//--------------------------------------------------------------------------------------------------------------------------------------------------------------------------------
3014://Comanda para posição de mesa de giro final após eixo X se movimentar 20% do trajeto para garantir que não colida a mesa de giro com a esteira de inspeção

	IF LA_GERAL.bit_MAQUINA_RODANDO AND (LA_EMP.info_MOTOR_EIXO_X_EMPILHADOR_POS_ATUAL > 130 AND LA_EMP.info_MOTOR_EIXO_X_EMPILHADOR_POS_ATUAL < 780) THEN
		LA_EMP.bit_EIXO_GIRO_MESA_MOVER_ABS		:= TRUE;
		
		passo_X_EMPILHADOR 									:= 3015;
	END_IF
	
//--------------------------------------------------------------------------------------------------------------------------------------------------------------------------------
3015: //verifica se a mesa de giro está se movendo para posição final. Caso esteja, desativa comando de movimento absoluto

	IF	M2_LA_EMP_GIRO.bit_MOVE_ABS_FAZENDO OR LA_EMP.bit_EIXO_GIRO_MESA_POSICIONADO	THEN
			LA_EMP.bit_EIXO_GIRO_MESA_MOVER_ABS	:= FALSE;
			passo_X_EMPILHADOR 								:= 3016;
	END_IF
	
//--------------------------------------------------------------------------------------------------------------------------------------------------------------------------------
3016: //verifica se a mesa de giro completou movimento

	IF	M2_LA_EMP_GIRO.bit_MOVE_ABS_FEITO OR LA_EMP.bit_EIXO_GIRO_MESA_POSICIONADO	THEN
			LA_EMP.bit_MESA_GIRO_CONCLUIDO	:= TRUE;
			passo_X_EMPILHADOR 							:= 3017;
	END_IF	
	
//--------------------------------------------------------------------------------------------------------------------------------------------------------------------------------
3017: //aguarda liberação da sacola depositada na mesa para liberar movimento do eixo X da empilhadora para próxima posição de pega	
	
// 	IF 		(PVAR.rec_ATUAL.int_NUM_MAX_CAMADAS_EMPILHADOR - 4) = 0 	THEN
// 				passo_X_EMPILHADOR			:= 3028;
// 	ELSIF 	(PVAR.rec_ATUAL.int_NUM_MAX_CAMADAS_EMPILHADOR - 4) = 1		THEN
// 				passo_X_EMPILHADOR			:= 3018;
// 		
// 	END_IF	

	IF 	(PVAR.rec_ATUAL.int_NUM_MAX_CAMADAS_EMPILHADOR - 4) = 0 	THEN
		M2_LA_EMP_GIRO.ABS_MOVER			:= PVAR.rec_ATUAL.coord_MESA_GIRO_INICIAL;
	END_IF

	passo_X_EMPILHADOR			:= 3018;
	
	
//--------------------------------------------------------------------------------------------------------------------------------------------------------------------------------
3018: //manda os valores de coordenada para movimentos absolutos da posição 9 do eixo X e declara que está na posição 9

	IF LA_EMP.bit_ENTREGA_EMPILHADOR_CONCLUIDO THEN
		M0_LA_EMP_X.ABS_MOVER	:= PVAR.rec_ATUAL.coord_X_EMPILHADOR_POS[PVAR.rec_ATUAL.int_NUM_MAX_CAMADAS_EMPILHADOR - 3];
		PVAR.int_POSICAO_EIXO_X_EMPILHADOR	:=	9;
		passo_X_EMPILHADOR 					:= 3019;
	END_IF
	
//--------------------------------------------------------------------------------------------------------------------------------------------------------------------------------
3019: // Comanda eixo X do empilhador com movimento absoluto para posição 9.

	IF LA_GERAL.bit_MAQUINA_RODANDO  THEN
		LA_EMP.bit_EIXO_X_EMPILHADOR_MOVER_ABS	:= TRUE;
		LA_EMP.bit_EIXO_GIRO_MESA_MOVER_ABS		:= TRUE;
		passo_X_EMPILHADOR 									:= 3020;	
	END_IF
	
//--------------------------------------------------------------------------------------------------------------------------------------------------------------------------------
3020: //verifica se o eixo X do empilhador está se movendo para posição 9. Caso esteja, desativa comando de movimento absoluto

	IF	M0_LA_EMP_X.bit_MOVE_ABS_FAZENDO OR LA_EMP.bit_EIXO_X_EMPILHADOR_POSICIONADO	THEN
			LA_EMP.bit_EIXO_X_EMPILHADOR_MOVER_ABS	:= FALSE;
			LA_EMP.bit_EIXO_GIRO_MESA_MOVER_ABS		:= FALSE;
			passo_X_EMPILHADOR 									:= 3021;
	END_IF
	
	
//--------------------------------------------------------------------------------------------------------------------------------------------------------------------------------
3021: //verifica se o eixo X do empilhador completou movimento

	IF	M0_LA_EMP_X.bit_MOVE_ABS_FEITO OR LA_EMP.bit_EIXO_X_EMPILHADOR_POSICIONADO	THEN
			LA_EMP.bit_LIBERA_PEGA			:= TRUE;
			passo_X_EMPILHADOR							:= 3022;
	END_IF


//--------------------------------------------------------------------------------------------------------------------------------------------------------------------------------
3022: //aguarda liberação da sacola depositada na mesa para liberar movimento do eixo X da empilhadora para POSIÇÃO 1

	IF 		(PVAR.rec_ATUAL.int_NUM_MAX_CAMADAS_EMPILHADOR - 4) = 0 		THEN
				passo_X_EMPILHADOR			:= 3025;
	ELSE		
				passo_X_EMPILHADOR			:= 3023;
	END_IF
	
//--------------------------------------------------------------------------------------------------------------------------------------------------------------------------------
3023: //manda os valores de coordenada para movimentos absolutos da posição 10 do eixo X e declara que está na posição 10

	IF LA_EMP.bit_ENTREGA_EMPILHADOR_CONCLUIDO THEN
		M0_LA_EMP_X.ABS_MOVER	:= PVAR.rec_ATUAL.coord_X_EMPILHADOR_POS[1];
		M2_LA_EMP_GIRO.ABS_MOVER			:= PVAR.rec_ATUAL.coord_MESA_GIRO_INICIAL;
		PVAR.int_POSICAO_EIXO_X_EMPILHADOR	:=	10;
		passo_X_EMPILHADOR 					:= 3024;
	END_IF
	
	// 	IF tmr_passo_3021.Q	THEN
	// 		passo_X_EMPILHADOR 					:= 3021;
	// 	END_IF
	
	
//--------------------------------------------------------------------------------------------------------------------------------------------------------------------------------
3024: // Comanda eixo X do empilhador com movimento absoluto para posição 10.

	IF LA_GERAL.bit_MAQUINA_RODANDO  THEN
		LA_EMP.bit_EIXO_X_EMPILHADOR_MOVER_ABS	:= TRUE;
		LA_EMP.bit_EIXO_GIRO_MESA_MOVER_ABS		:= TRUE;
		passo_X_EMPILHADOR 									:= 3025;	
	END_IF
	
//--------------------------------------------------------------------------------------------------------------------------------------------------------------------------------
3025: //verifica se o eixo X do empilhador está se movendo para posição 10. Caso esteja, desativa comando de movimento absoluto

	IF	M0_LA_EMP_X.bit_MOVE_ABS_FAZENDO OR LA_EMP.bit_EIXO_X_EMPILHADOR_POSICIONADO	THEN
			LA_EMP.bit_EIXO_X_EMPILHADOR_MOVER_ABS	:= FALSE;
			passo_X_EMPILHADOR 									:= 3026;
	END_IF
	
//--------------------------------------------------------------------------------------------------------------------------------------------------------------------------------
3026: //verifica se o eixo rotativo do empilhador está se movendo para posição inicial. Caso esteja, desativa comando de movimento absoluto

	IF	M2_LA_EMP_GIRO.bit_MOVE_ABS_FAZENDO OR LA_EMP.bit_EIXO_GIRO_MESA_POSICIONADO	THEN
			LA_EMP.bit_EIXO_GIRO_MESA_MOVER_ABS		:= FALSE;
			passo_X_EMPILHADOR 									:= 3027;
	END_IF
	
//--------------------------------------------------------------------------------------------------------------------------------------------------------------------------------
3027: //verifica se o eixo X do empilhador completou movimento	
	
	IF	M0_LA_EMP_X.bit_MOVE_ABS_FEITO	OR 	LA_EMP.bit_EIXO_X_EMPILHADOR_POSICIONADO	THEN
			bit_X_EMPILHADOR_FEITO				:= TRUE;
			LA_EMP.bit_LIBERA_PEGA	:= TRUE;
	END_IF	
	
	IF	M2_LA_EMP_GIRO.bit_MOVE_ABS_FEITO	OR 	LA_EMP.bit_EIXO_GIRO_MESA_POSICIONADO	THEN
			bit_GIRO_MESA_FEITO	:= TRUE;
	END_IF	
	
	IF	bit_X_EMPILHADOR_FEITO		AND
		bit_GIRO_MESA_FEITO			THEN
			bit_X_EMPILHADOR_FEITO		:= FALSE;
			bit_GIRO_MESA_FEITO			:= FALSE;
		
			passo_X_EMPILHADOR 			:= 3028;
	END_IF		
	
//--------------------------------------------------------------------------------------------------------------------------------------------------------------------------------
3028://aguarda confirmação de pilha entregue e comanda posições para entregar pilha para inspeção

	M0_LA_EMP_X.ABS_MOVER		 	:= PVAR.rec_ATUAL.coord_X_EMPILHADOR_INSPECAO;
	M2_LA_EMP_GIRO.ABS_MOVER		 			:= PVAR.rec_ATUAL.coord_MESA_GIRO_INSPECAO;
	LA_EMP.bit_REALIZANDO_INSPECAO 	:= TRUE;
	passo_X_EMPILHADOR							:= 3029;
	
//--------------------------------------------------------------------------------------------------------------------------------------------------------------------------------
3029://comanda movimento da mesa de giro para posição de inspeção

	LA_EMP.bit_LIBERA_PEGA	:= FALSE;

	IF LA_GERAL.bit_MAQUINA_RODANDO AND LA_EMP.bit_ENTREGA_EMPILHADOR_CONCLUIDO	THEN
		LA_EMP.bit_EIXO_GIRO_MESA_MOVER_ABS		:= TRUE;
		passo_X_EMPILHADOR									:= 3030;
	END_IF

//--------------------------------------------------------------------------------------------------------------------------------------------------------------------------------
3030: //verifica se o eixo rotativo do empilhador está se movendo para posição inicial. Caso esteja, desativa comando de movimento absoluto

	IF	M2_LA_EMP_GIRO.bit_MOVE_ABS_FAZENDO OR LA_EMP.bit_EIXO_GIRO_MESA_POSICIONADO	THEN
			LA_EMP.bit_EIXO_GIRO_MESA_MOVER_ABS		:= FALSE;
			passo_X_EMPILHADOR 									:= 3031;
	END_IF	
	
//--------------------------------------------------------------------------------------------------------------------------------------------------------------------------------
3031://verifica se a mesa de giro completou o movimento	

	IF	M2_LA_EMP_GIRO.bit_MOVE_ABS_FEITO OR LA_EMP.bit_EIXO_GIRO_MESA_POSICIONADO	THEN
			passo_X_EMPILHADOR 	:= 3032;
	END_IF

//--------------------------------------------------------------------------------------------------------------------------------------------------------------------------------
3032://se a máquina estiver rodando, comanda movimento do eixo X do empilhador para inspeção

	IF LA_GERAL.bit_MAQUINA_RODANDO	THEN
		LA_EMP.bit_EIXO_X_EMPILHADOR_MOVER_ABS	:= TRUE;
		passo_X_EMPILHADOR 									:= 3033;
	END_IF
	
//--------------------------------------------------------------------------------------------------------------------------------------------------------------------------------
3033://verifica se o eixo X do empilhador está se movendo para inspeção. Caso esteja, desativa comando de movimento absoluto

	IF	M0_LA_EMP_X.bit_MOVE_ABS_FAZENDO OR LA_EMP.bit_EIXO_X_EMPILHADOR_POSICIONADO	THEN
			LA_EMP.bit_EIXO_X_EMPILHADOR_MOVER_ABS	:= FALSE;
			passo_X_EMPILHADOR 									:= 3034;
	END_IF	
	
//--------------------------------------------------------------------------------------------------------------------------------------------------------------------------------
3034: // verifica se eixo X do empilhador completou movimento

	IF	M0_LA_EMP_X.bit_MOVE_ABS_FEITO OR  LA_EMP.bit_EIXO_X_EMPILHADOR_POSICIONADO	THEN
		LA_EMP.bit_LIBERA_INSPECAO_PILHA		:= 	TRUE;
		passo_X_EMPILHADOR 								:= 3035;
	END_IF	

	
//--------------------------------------------------------------------------------------------------------------------------------------------------------------------------------
3035://liga esteira de mesa giro para liberar pilha de sacola para esteira de inspeção
	
	LA_EMP.est_ROLETES_GIRO_MESA_REVERSE	:= FALSE;
	LA_EMP.est_ROLETES_GIRO_MESA			:= TRUE;
	passo_X_EMPILHADOR 								:= 3036;
	
//--------------------------------------------------------------------------------------------------------------------------------------------------------------------------------
3036://Após um tempo fora do sensor de presença da mesa de giro, considera que a pilha saiu da mesa de giro e conclui processo de entrega para mesa de inspeção
	

	IF LA_EMP.di_SENS_EST_INSPEC_PRODUTO_2 AND NOT LA_EMP.di_SENS_PRODUTO_MESA_GIRO THEN
		bit_RESET_CONTAGEM		:= TRUE;
		passo_X_EMPILHADOR 		:= 3037;
	END_IF
	
	
//--------------------------------------------------------------------------------------------------------------------------------------------------------------------------------
3037://Declara pilha como entregue e para a esteira da mesa giro. Prepara mesa de giro para posição de reinicio

	tmr_sens_MESA_GIRO_IN.IN						:= FALSE;
	LA_EMP.est_ROLETES_GIRO_MESA			:= FALSE;
	LA_EMP.est_ROLETES_GIRO_MESA_REVERSE	:= FALSE;
	
	LA_EMP.bit_EST_PILHA_ENTREGUE		 	:= FALSE;
	LA_EMP.bit_LIBERA_INSPECAO_PILHA	 	:= FALSE;
	LA_EMP.bit_EST_INSPECAO_ENTREGUE_1 	:= FALSE;
	LA_EMP.bit_EST_INSPECAO_ENTREGUE_2 	:= FALSE;
	bit_RESET_CONTAGEM							 	:= FALSE;
	LA_EMP.bit_REALIZANDO_INSPECAO	 	:= FALSE;
	LA_EMP.bit_valv_DESCE_MESA_GIRO	 	:= FALSE;

	passo_X_EMPILHADOR							 	:= 998;
	

	
END_CASE

//--------------------------------------------------------------------------------------------------------------------------------------------------------------------------------
//--------------------------------------------------------------------------------------------------------------------------------------------------------------------------------
//LÓGICAS AUXILIARES


	
	
(*//CONTINUAR MOVIMENTO DO EIXO X DO EMPILHADOR APÓS PARADA DE EMERGÊNCIA
	IF (bt_MAQUINA_RESET OR bt_MAQUINA_RESET_2) AND NOT GVL_CELULA.bit_MAQUINA_RODANDO	THEN
			
			IF 	passo_X_EMPILHADOR >= 0 	AND
				passo_X_EMPILHADOR <= 15 	THEN
				GVL_EMPILHAMENTO.bit_EIXO_X_EMPILHADOR_MOVER_ABS		:= FALSE;
				passo_X_EMPILHADOR := 9;
			END_IF	
	
			IF 	(passo_X_EMPILHADOR >= 1000	AND
				passo_X_EMPILHADOR <= 1003) THEN
				GVL_EMPILHAMENTO.bit_EIXO_X_EMPILHADOR_MOVER_ABS		:= FALSE;
				passo_X_EMPILHADOR := 999;
			END_IF
			
			IF 	passo_X_EMPILHADOR >= 1005 	AND
				passo_X_EMPILHADOR <= 1008 	THEN
				GVL_EMPILHAMENTO.bit_EIXO_X_EMPILHADOR_MOVER_ABS		:= FALSE;
				passo_X_EMPILHADOR := 1005;
			END_IF
			
			IF 	passo_X_EMPILHADOR >= 1010 	AND
				passo_X_EMPILHADOR <= 1013 	THEN
				GVL_EMPILHAMENTO.bit_EIXO_X_EMPILHADOR_MOVER_ABS		:= FALSE;
				passo_X_EMPILHADOR := 1010;
			END_IF
			
			IF 	passo_X_EMPILHADOR >= 1015 	AND
				passo_X_EMPILHADOR <= 1018 	THEN
				GVL_EMPILHAMENTO.bit_EIXO_X_EMPILHADOR_MOVER_ABS		:= FALSE;
				passo_X_EMPILHADOR := 1015;
			END_IF
			
			IF 	passo_X_EMPILHADOR >= 1020 	AND
				passo_X_EMPILHADOR <= 1023 	THEN
				GVL_EMPILHAMENTO.bit_EIXO_X_EMPILHADOR_MOVER_ABS		:= FALSE;
				passo_X_EMPILHADOR := 1020;
			END_IF
			
			IF 	passo_X_EMPILHADOR >= 1025 	AND
				passo_X_EMPILHADOR <= 1028 	THEN
				GVL_EMPILHAMENTO.bit_EIXO_X_EMPILHADOR_MOVER_ABS		:= FALSE;
				passo_X_EMPILHADOR := 1025;
			END_IF
			
			IF 	passo_X_EMPILHADOR >= 2000 	AND
				passo_X_EMPILHADOR <= 2003	THEN
				GVL_EMPILHAMENTO.bit_EIXO_X_EMPILHADOR_MOVER_ABS		:= FALSE;
				passo_X_EMPILHADOR := 2000;
			END_IF
			
			IF 	passo_X_EMPILHADOR >= 2005 	AND
				passo_X_EMPILHADOR <= 2008	THEN
				GVL_EMPILHAMENTO.bit_EIXO_X_EMPILHADOR_MOVER_ABS		:= FALSE;
				passo_X_EMPILHADOR := 2005;
			END_IF
			
			IF 	passo_X_EMPILHADOR >= 2010 	AND
				passo_X_EMPILHADOR <= 2013	THEN
				GVL_EMPILHAMENTO.bit_EIXO_X_EMPILHADOR_MOVER_ABS		:= FALSE;
				passo_X_EMPILHADOR := 2010;
			END_IF
			
			IF 	passo_X_EMPILHADOR >= 2015 	AND
				passo_X_EMPILHADOR <= 2015	THEN
				GVL_EMPILHAMENTO.bit_EIXO_X_EMPILHADOR_MOVER_ABS		:= FALSE;
				passo_X_EMPILHADOR := 2015;
			END_IF
			
			IF 	passo_X_EMPILHADOR >= 2020 	AND
				passo_X_EMPILHADOR <= 2023	THEN
				GVL_EMPILHAMENTO.bit_EIXO_X_EMPILHADOR_MOVER_ABS		:= FALSE;
				passo_X_EMPILHADOR := 2020;
			END_IF
			
	END_IF
	
*)

	
	
	//EIXO X EMPILHADOR JÁ ESTÁ NA POSIÇÃO
	IF	LA_EMP.info_MOTOR_EIXO_X_EMPILHADOR_POS_ATUAL	>= M0_LA_EMP_X.ABS_MOVER.sp_POSICAO - 1	AND
		LA_EMP.info_MOTOR_EIXO_X_EMPILHADOR_POS_ATUAL	<= M0_LA_EMP_X.ABS_MOVER.sp_POSICAO + 1	THEN
			LA_EMP.bit_EIXO_X_EMPILHADOR_POSICIONADO	:= TRUE;
	ELSE
			LA_EMP.bit_EIXO_X_EMPILHADOR_POSICIONADO	:= FALSE;
	END_IF
	
	
	//EIXO X EMPILHADOR JÁ ESTÁ NA POSIÇÃO
	IF	LA_EMP.info_MOTOR_GIRO_MESA_POS_ATUAL	>= M2_LA_EMP_GIRO.ABS_MOVER.sp_POSICAO - 1	AND
		LA_EMP.info_MOTOR_GIRO_MESA_POS_ATUAL	<= M2_LA_EMP_GIRO.ABS_MOVER.sp_POSICAO + 1	THEN
			LA_EMP.bit_EIXO_GIRO_MESA_POSICIONADO	:= TRUE;
	ELSE
			LA_EMP.bit_EIXO_GIRO_MESA_POSICIONADO	:= FALSE;
	END_IF
	
	
		
	//Define se a posicão da mesa de giro de acordo com a posição atual do eixo X
	IF M2_LA_EMP_GIRO.ABS_MOVER.sp_POSICAO > 90 THEN
		LA_EMP.bit_GIRO_MESA_FOWARD	:=	TRUE;
		LA_EMP.bit_GIRO_MESA_REVERSE	:=	FALSE;
	ELSE
		LA_EMP.bit_GIRO_MESA_FOWARD	:=	FALSE;
		LA_EMP.bit_GIRO_MESA_REVERSE	:=	TRUE;
	END_IF
	

	
	
//TIMERS EIXO X
tmr_HOME 	  (PT	:= T#200MS);
tmr_ENTREGA_X (PT	:= T#100MS);
tmr_passo_2021(PT	:= T#300MS);
tmr_passo_2032(PT	:= T#500MS);
tmr_LIBERA_X_INSPECAO(PT	:= T#1500MS);
cont_PILHA_ENTREGA(CU:= bit_INCREMENTA_SACOLA, RESET:= bit_RESET_CONTAGEM, PV:= 999, CV=> pvar.int_PILHAS_ENTREGUES);	


//TIMERS GIRO MESA
tmr_HOME 			(PT	:= T#200MS);
tmr_sens_MESA_GIRO_IN 	(PT	:= T#500MS);
tmr_sens_MESA_GIRO_OUT 	(PT	:= T#2300MS);
TMR_GIRO_1		 	(PT	:= T#4000MS);
TMR_GIRO_2		 	(PT	:= T#4000MS);
TMR_GIRO_3		 	(PT	:= T#4000MS);
TMR_GIRO_4		 	(PT	:= T#500MS);
TMR_GIRO_5		 	(PT	:= T#4000MS);
TMR_GIRO_10		 	(PT	:= T#4000MS);

tmr_passo_1041		 	(PT	:= T#300MS);

END_PROGRAM

// LADO_A/02 - LA_EMPILHADOR/B03_INSPECAO
PROGRAM B03_INSPECAO
VAR
	passo_INSPECAO		: INT := 9;
	tmr_INSPECAO_OK		: TON;
	tmr_LIBERA_INSPECAO_OK		: TON;
END_VAR

//MOVE O PASSO PARA O HOME

	IF	LA_IHM.bit_bt_RESET_INSPECAO	THEN
			passo_INSPECAO								:= 9;
	END_IF
	
CASE	passo_INSPECAO	OF
	
//--------------------------------------------------------------------------------------------------------------------------------------------------------------------------------
09: //HOME: Reseta variáveis

	IF NOT LA_EMP.di_SENS_EST_INSPEC_PRODUTO_1 AND NOT LA_EMP.di_SENS_EST_INSPEC_PRODUTO_2 THEN
		LA_EMP.bit_OPERADOR_INSPECAO_OK		:=	FALSE;
		LA_EMP.bit_EST_ENVIAR_PILHA_INSPECAO	:=	FALSE;
		LA_EMP.bit_EST_INSPECAO_ENTREGUE_2	:=	FALSE;
		LA_EMP.est_INSPECAO_EMPILHADOR		:= 	FALSE;
		tmr_LIBERA_INSPECAO_OK.IN						:=	FALSE;
		bt_LAMP_INSPECAO_OK 							:=  FALSE;
		passo_INSPECAO									:=  999;
	ELSIF LA_EMP.bit_OPERADOR_INSPECAO_OK THEN
		passo_INSPECAO									:= 1002;
	END_IF
	
	
//--------------------------------------------------------------------------------------------------------------------------------------------------------------------------------
999://aguarda esteira da mesa giro entregar pilha para inspeção e liga esteira

	IF LA_EMP.bit_LIBERA_INSPECAO_PILHA	THEN
		LA_EMP.est_INSPECAO_EMPILHADOR	:= TRUE;
		passo_INSPECAO								:= 1000;
	END_IF
	
	IF LA_EMP.bit_OPERADOR_INSPECAO_OK THEN
		LA_EMP.bit_STATUS_INSPECAO_1		:= FALSE;
		passo_INSPECAO								:= 1002;
	END_IF
	
	
//--------------------------------------------------------------------------------------------------------------------------------------------------------------------------------
1000://espera feedback dos sensores da esteira de inspeção para garantir que a pilha chegou até o fim. 

	IF  LA_EMP.di_SENS_EST_INSPEC_PRODUTO_2 THEN
		LA_EMP.est_INSPECAO_EMPILHADOR		:= FALSE;
		LA_EMP.bit_STATUS_INSPECAO_1			:= TRUE;
		//GVL_EMPILHAMENTO.bit_EST_INSPECAO_ENTREGUE_1	:= TRUE;
		
		passo_INSPECAO									:= 999;
	END_IF
	
	
//--------------------------------------------------------------------------------------------------------------------------------------------------------------------------------
1001://aguarda comando de operador indicando que a pilha está ok para ser devolvida

	IF LA_EMP.bit_OPERADOR_INSPECAO_OK THEN
		LA_EMP.bit_STATUS_INSPECAO_1	:= FALSE;
		passo_INSPECAO							:= 1002;
	END_IF
	
//--------------------------------------------------------------------------------------------------------------------------------------------------------------------------------
1002://espera confirmação de recebimento OK da esteira mesa giro e liga esteira de inspeção reverse para devolução de pilha 

	IF LA_EMP.bit_EST_ENVIAR_PILHA_INSPECAO THEN
		LA_EMP.est_INSPECAO_EMPILHADOR_REVERSE 	:= TRUE;
		LA_EMP.est_INSPECAO_EMPILHADOR			:= TRUE;
		passo_INSPECAO										:= 1003;
	END_IF
	
	
//--------------------------------------------------------------------------------------------------------------------------------------------------------------------------------
1003://ao deixar de receber feedback dos dois sensores da esteira de inspeção, para esteira e reinicia ciclo

	IF NOT LA_EMP.di_SENS_EST_INSPEC_PRODUTO_1 AND NOT LA_EMP.di_SENS_EST_INSPEC_PRODUTO_2 THEN
		tmr_LIBERA_INSPECAO_OK.IN							:= TRUE;
	ELSE
		tmr_LIBERA_INSPECAO_OK.IN							:= FALSE;
	END_IF
	
	IF tmr_LIBERA_INSPECAO_OK.Q	THEN
		passo_INSPECAO										:= 1004;
	END_IF
	
//--------------------------------------------------------------------------------------------------------------------------------------------------------------------------------
1004:
		LA_EMP.est_INSPECAO_EMPILHADOR_REVERSE	:= FALSE;
		LA_EMP.est_INSPECAO_EMPILHADOR			:= FALSE;
		tmr_LIBERA_INSPECAO_OK.IN							:= FALSE;
		LA_EMP.bit_EST_INSPECAO_ENTREGUE_2		:= TRUE;
		passo_INSPECAO										:= 999;

END_CASE




//------------LÓGICAS ADICIONAIS-------------------//--------------------------------------//---------------------------------

	//LIBERAÇÃO DE PILHA DE INSPEÇÃO COMO OK AO DETECTAR PILHA NOS SENSORES DA ESTEIRA DE INSPEÇÃO
	IF tmr_INSPECAO_OK.Q AND (LA_EMP.di_SENS_EST_INSPEC_PRODUTO_2)	THEN
		LA_EMP.bit_OPERADOR_INSPECAO_OK	:=	TRUE;
	END_IF

	IF NOT LA_EMP.bit_STATUS_INSPECAO_1 AND NOT LA_EMP.bit_OPERADOR_INSPECAO_OK THEN
		LA_IHM.bit_STATUS_INSPECAO_OK	:=	0;
	ELSIF LA_EMP.bit_STATUS_INSPECAO_1 AND NOT LA_EMP.bit_OPERADOR_INSPECAO_OK THEN
		LA_IHM.bit_STATUS_INSPECAO_OK	:=	1;
	ELSIF LA_EMP.bit_OPERADOR_INSPECAO_OK	THEN
		LA_IHM.bit_STATUS_INSPECAO_OK	:=	2;
	END_IF

//TIMERS
tmr_INSPECAO_OK(IN:= bt_INSPECAO_OK OR LA_IHM.bit_bt_INSPECAO_OK, PT:= T#2S );
tmr_LIBERA_INSPECAO_OK(PT:= T#2S );

END_PROGRAM

// LADO_A/02 - LA_EMPILHADOR/B04_ENTRADAS_REMOTAS
PROGRAM B04_ENTRADAS_REMOTAS
VAR
END_VAR


//	SLOT 1		============//============//============//============//============//============//============

	LA_EMP.di_SENS_MESA_GIRO_RC					:= di_LOCAL_SLOT1_0;
	
	LA_EMP.di_SENS_MESA_GIRO_MD					:= di_LOCAL_SLOT1_1;
	
	LA_EMP.di_SENS_PINCA_GARRA_EMPILHADOR_RC	:= di_LOCAL_SLOT1_2;
	
	LA_EMP.di_SENS_APOIO_BANDEJA_RC				:= di_LOCAL_SLOT1_3;
	
	//											:= di_LOCAL_SLOT1_4;
	
	LA_EMP.di_SENS_EST_INSPEC_PRODUTO_1			:= di_LOCAL_SLOT1_5;
	
	//RESERVA									:= di_LOCAL_SLOT1_6;
	
	//RESERVA									:= di_LOCAL_SLOT1_7;
	
	LA_EMP.di_SENS_MESA_GIRO_AV					:= di_LOCAL_SLOT1_8;
	
	//											:= di_LOCAL_SLOT1_9;
	
	LA_EMP.di_SENS_PINCA_GARRA_EMPILHADOR_AV	:= di_LOCAL_SLOT1_10;
	
	LA_EMP.di_SENS_APOIO_BANDEJA_AV				:= di_LOCAL_SLOT1_11;
	
	LA_EMP.di_SENS_PRODUTO_MESA_GIRO			:= di_LOCAL_SLOT1_12;
	
	LA_EMP.di_SENS_EST_INSPEC_PRODUTO_2			:= di_LOCAL_SLOT1_13;
	
	//											:= di_LOCAL_SLOT1_14;
	
	//											:= di_LOCAL_SLOT1_15;
	
	
//	SLOT 2		============//============//============//============//============//============//============

	LA_EMP.di_feedback_ERRO_MESA_GIRO			:= di_REMOTA_SLOT2_10;
	
	LA_EMP.di_feedback_ERRO_EST_INSPECAO		:= di_REMOTA_SLOT2_12;

END_PROGRAM

// LADO_A/02 - LA_EMPILHADOR/B05_SAIDAS_REMOTAS
PROGRAM B05_SAIDAS_REMOTAS
VAR
END_VAR

//	SLOT 1		============//============//============//============//============//============//============
	
	do_REMOTA_SLOT1_6	:= LA_EMP.do_ATU_MESA_GIRO_RC;
	
	do_REMOTA_SLOT1_7	:= LA_EMP.do_ATU_PINCA_GARRA_EMPILHADOR;
	
	do_REMOTA_SLOT1_16	:= LA_EMP.do_ATU_MESA_GIRO_AV;
	
	do_REMOTA_SLOT1_17	:= LA_EMP.do_ATU_BANDEJA_APOIO;

END_PROGRAM

// LADO_A/03 - LA_ENVOLVEDOR/C01_GIRO_SACOLA
PROGRAM C01_GIRO_SACOLA
VAR
	passo_GIRO_SACOLA			: INT := 9;
	
	bit_ENTREGA_X_FEITO			: BOOL;
	bit_ENTREGA_GIRO_LD_FEITO	: BOOL;
	bit_ENTREGA_GIRO_LE_FEITO	: BOOL;
	
	bit_MOVE_REL_GIRO_GARRA		: BOOL;
	
	tmr_APROX_GARRA				: TON;
	tmr_GARRA_DUPLA				: TON;
	tmr_GARRA_DUPLA2			: TON;
	tmr_GARRA_DUPLA3			: TON;
	tmr_GARRA_DUPLA4			: TON;
	
	tmr_FECHA_FILME_1			: TON;
	
	tmr_PASSO_1028				: TON;
	tmr_PASSO_1029				: TON;
END_VAR

	IF LA_IHM.bit_GIRO_SACOLA_RESET THEN
		passo_GIRO_SACOLA	:=	9;
	END_IF
	
CASE passo_GIRO_SACOLA OF
	

//--------------------------------------------------------------------------------------------------------------------------------------------------------------------------------
09: //HOME: Reseta variáveis
	
	LA_ENV.bit_EIXO_Z_ENVOLVEDOR_FAZER_HOME			:= FALSE;
	LA_ENV.bit_EIXO_Z_ENVOLVEDOR_MOVER_ABS			:= FALSE;
	M3_LA_ENV_Z.bit_FAZER_HOME				:= FALSE;
	
	LA_ENV.bit_EIXO_X_ENVOLVEDOR_FAZER_HOME			:= FALSE;
	LA_ENV.bit_EIXO_X_ENVOLVEDOR_MOVER_ABS			:= FALSE;
	M4_LA_ENV_X.bit_FAZER_HOME				:= FALSE;
	
	LA_ENV.bit_EIXO_GIRO_ENVOLVEDOR_LD_FAZER_HOME	:= FALSE;
	LA_ENV.bit_EIXO_GIRO_ENVOLVEDOR_LD_MOVER_ABS	:= FALSE;
	
	LA_ENV.bit_EIXO_GIRO_ENVOLVEDOR_LE_FAZER_HOME	:= FALSE;
	LA_ENV.bit_EIXO_GIRO_ENVOLVEDOR_LE_MOVER_ABS	:= FALSE;
	
	bit_ENTREGA_X_FEITO			:= FALSE;
	bit_ENTREGA_GIRO_LD_FEITO	:= FALSE;
	bit_ENTREGA_GIRO_LE_FEITO	:= FALSE;
	
	LA_ENV.bit_ENV_CORTE_FILME	:= FALSE;
	LA_ENV.bit_valv_VACUO_FILME	:=	TRUE;
	
	
	LA_ENV.bit_ENVOLVEDOR_SACOLA_DEPOSITANDO		:=	FALSE;
	
	tmr_PASSO_1028.IN					:=	FALSE;
	tmr_PASSO_1029.IN					:=	FALSE;
	
	passo_GIRO_SACOLA						:= 10;
	
//--------------------------------------------------------------------------------------------------------------------------------------------------------------------------------
10: //HOME: Se a máquina estiver rodando e não estiver em modo manual, começa o processo de Home
	
	IF LA_GERAL.bit_MAQUINA_PRONTA  THEN
			LA_ENV.bit_valv_GARRA_DUPLA		:=	FALSE;
		
			passo_GIRO_SACOLA	:= 11;
	END_IF
	
	
//--------------------------------------------------------------------------------------------------------------------------------------------------------------------------------
11: //HOME: Inicia o Home no eixo Z do Envolvedor
	
	LA_ENV.bit_EIXO_Z_ENVOLVEDOR_FAZER_HOME		:= TRUE;

	passo_GIRO_SACOLA									:= 13;
	
//--------------------------------------------------------------------------------------------------------------------------------------------------------------------------------
13: //HOME: Verifica se está se movendo para o Home do Eixo Z do Envolvedor
	
	IF M3_LA_ENV_Z.bit_HOME_FAZENDO	THEN
			
			passo_GIRO_SACOLA					:= 14;
	END_IF
	

//--------------------------------------------------------------------------------------------------------------------------------------------------------------------------------
14: //HOME: Se o Home do eixo Z do Envolvedor for concluído, vai para próximo passo. 

	IF	M3_LA_ENV_Z.bit_HOME_FEITO	THEN
			M3_LA_ENV_Z.bit_FAZER_HOME					:= FALSE;
			LA_ENV.bit_valv_APROX_GARRA				:=	TRUE;
			LA_ENV.bit_EIXO_Z_ENVOLVEDOR_FAZER_HOME	:= FALSE;
			passo_GIRO_SACOLA										:= 15;
	END_IF
	
	
//--------------------------------------------------------------------------------------------------------------------------------------------------------------------------------
15: //HOME: Inicia o Home no eixo X do Envolvedor
	
	IF	LA_GERAL.di_ENV_SENS_ATU_ABERTURA_AV	THEN
		LA_ENV.bit_EIXO_X_ENVOLVEDOR_FAZER_HOME		:= TRUE;
		passo_GIRO_SACOLA									:= 16;
	END_IF
	
	
//--------------------------------------------------------------------------------------------------------------------------------------------------------------------------------
16: //HOME: Verifica se está se movendo para o Home do Eixo X do Envolvedor
	
	IF M4_LA_ENV_X.bit_HOME_FAZENDO	THEN
			
			passo_GIRO_SACOLA					:= 17;
	END_IF
	

//--------------------------------------------------------------------------------------------------------------------------------------------------------------------------------
17: //HOME: Se o Home do eixo X do Envolvedor for concluído, vai para próximo passo. 

	IF	M4_LA_ENV_X.bit_HOME_FEITO	THEN
			M4_LA_ENV_X.bit_FAZER_HOME					:= FALSE;
			LA_ENV.bit_EIXO_X_ENVOLVEDOR_FAZER_HOME	:= FALSE;
			passo_GIRO_SACOLA										:= 18;
	END_IF

	
//--------------------------------------------------------------------------------------------------------------------------------------------------------------------------------
18: //HOME: Inicia o Home no eixos de giro do Envolvedor
	
	LA_ENV.bit_EIXO_GIRO_ENVOLVEDOR_LD_FAZER_HOME		:= TRUE;
	LA_ENV.bit_EIXO_GIRO_ENVOLVEDOR_LE_FAZER_HOME		:= TRUE;

	passo_GIRO_SACOLA							:= 19;
	
//--------------------------------------------------------------------------------------------------------------------------------------------------------------------------------
19: //HOME: Verifica se está se movendo para o Home dos eixos de giro do Envolvedor
	
	IF M5_LA_ENV_GIRO_LD.bit_HOME_FAZENDO AND M6_LA_ENV_GIRO_LE.bit_HOME_FAZENDO	THEN
			LA_ENV.bit_EIXO_GIRO_ENVOLVEDOR_LD_FAZER_HOME	:= FALSE;
			LA_ENV.bit_EIXO_GIRO_ENVOLVEDOR_LE_FAZER_HOME	:= FALSE;
			passo_GIRO_SACOLA					:= 20;
	END_IF
		
//--------------------------------------------------------------------------------------------------------------------------------------------------------------------------------
20: //HOME: Se o Home dos eixos do Envolvedor forem concluído, vai para próximo passo. Se não, reinicia o home de novo
	
	IF	M5_LA_ENV_GIRO_LD.bit_HOME_FEITO AND M6_LA_ENV_GIRO_LE.bit_HOME_FEITO	THEN
			passo_GIRO_SACOLA						:= 100;
	END_IF
	
//--------------------------------------------------------------------------------------------------------------------------------------------------------------------------------
100: //HOME:
	IF LA_GERAL.bit_MAQUINA_RODANDO THEN
		passo_GIRO_SACOLA	:=	101;
	END_IF
	

//--------------------------------------------------------------------------------------------------------------------------------------------------------------------------------
101: //HOME: resetando atuadores

	 passo_GIRO_SACOLA	:=	102;
	IF	LA_GERAL.di_ENV_SENS_ATU_ABERTURA_RC 	THEN
			passo_GIRO_SACOLA	:=	102;
	END_IF
	
//--------------------------------------------------------------------------------------------------------------------------------------------------------------------------------
102://HOME: resetando atuadores
	
		passo_GIRO_SACOLA	:=	999;

	
//--------------------------------------------------------------------------------------------------------------------------------------------------------------------------------
999://SE A MÁQUINA ESTIVER RODANDO, PREPARA INICIO DE CICLO

	IF LA_GERAL.bit_MAQUINA_RODANDO THEN
		passo_GIRO_SACOLA	:=	1000;	
	END_IF
	
//--------------------------------------------------------------------------------------------------------------------------------------------------------------------------------
1000://	comanda posição de pega dos eixo X, LD e LE do envolvedor

	M4_LA_ENV_X.ABS_MOVER		:= LA_GERAL.coord_X_ENVOLVEDOR_PEGA;
	
	passo_GIRO_SACOLA 						:= 1001;
	
//--------------------------------------------------------------------------------------------------------------------------------------------------------------------------------
1001: //Comanda eixos X e rotativos do Envolvedor com movimentos absolutos para ponto de pega de filme. 

	LA_ENV.bit_EIXO_X_ENVOLVEDOR_MOVER_ABS				:= TRUE;
	LA_ENV.bit_valv_GARRA_DUPLA				 			:= FALSE;
		
	passo_GIRO_SACOLA 		:= 1002;
	
//--------------------------------------------------------------------------------------------------------------------------------------------------------------------------------
1002: //Verifica se Eixo X do envolvedor está se movimentando ou se já está posicionado

	IF	M4_LA_ENV_X.bit_MOVE_ABS_FAZENDO	OR 	LA_ENV.bit_EIXO_X_ENVOLVEDOR_POSICIONADO	THEN
			LA_ENV.bit_EIXO_X_ENVOLVEDOR_MOVER_ABS	:= FALSE;
			passo_GIRO_SACOLA 								:= 1003;
	END_IF
	
//--------------------------------------------------------------------------------------------------------------------------------------------------------------------------------
1003: //Verifica se Eixo LD do envolvedor está se movimentando ou se já está posicionado

			passo_GIRO_SACOLA 				:= 1004;
	
//--------------------------------------------------------------------------------------------------------------------------------------------------------------------------------
1004: //Verifica se Eixo LE do envolvedor está se movimentando ou se já está posicionado

			passo_GIRO_SACOLA 				:= 1005;
	
//--------------------------------------------------------------------------------------------------------------------------------------------------------------------------------
1005: //verifica se Eixos LD, LE e X chegaram aos seus pontos

	IF	M4_LA_ENV_X.bit_MOVE_ABS_FEITO	OR 	LA_ENV.bit_EIXO_X_ENVOLVEDOR_POSICIONADO	THEN
			passo_GIRO_SACOLA 			:= 1006;
	END_IF	
			
//--------------------------------------------------------------------------------------------------------------------------------------------------------------------------------
1006://	comanda posição de pre pega do eixo Z do envolvedor

	IF 	LA_GERAL.bit_MAQUINA_RODANDO 				THEN
			M3_LA_ENV_Z.ABS_MOVER	:= 	LA_GERAL.coord_Z_ENVOLVEDOR_PRE_PEGA;
			passo_GIRO_SACOLA					:=	1007;
	END_IF
		
//--------------------------------------------------------------------------------------------------------------------------------------------------------------------------------
1007://se estiver rodando, libera movimento do eixo Z do Envolvedor

	IF LA_GERAL.bit_MAQUINA_RODANDO THEN
		LA_ENV.bit_EIXO_Z_ENVOLVEDOR_MOVER_ABS	:= TRUE;
		passo_GIRO_SACOLA								:= 1008;	
	END_IF
	
//--------------------------------------------------------------------------------------------------------------------------------------------------------------------------------
1008://verifica se eixo Z do Envolvedor está se movendo ou se já está posicionado

	IF	M3_LA_ENV_Z.bit_MOVE_ABS_FAZENDO OR LA_ENV.bit_EIXO_Z_ENVOLVEDOR_POSICIONADO	THEN
		LA_ENV.bit_EIXO_Z_ENVOLVEDOR_MOVER_ABS	:= FALSE;
		
		passo_GIRO_SACOLA								:= 1009;
	END_IF
	
//--------------------------------------------------------------------------------------------------------------------------------------------------------------------------------
1009://verifica se eixo Z do Envolvedor completou movimento

	IF	M3_LA_ENV_Z.bit_MOVE_ABS_FEITO OR LA_ENV.bit_EIXO_Z_ENVOLVEDOR_POSICIONADO	THEN
		LA_ENV.bit_EIXO_Z_ENVOLVEDOR_MOVER_ABS	:= FALSE;
		LA_ENV.bit_valv_APROX_GARRA				:=	false;
		
		passo_GIRO_SACOLA					:= 1010;
	END_IF
	
//--------------------------------------------------------------------------------------------------------------------------------------------------------------------------------
1010://	comanda posição de pega do eixo Z do envolvedor a sacola e o strech estejam posicionados

	IF 	LA_GERAL.bit_MAQUINA_RODANDO 					AND
		LA_ENV.bit_ENVOLVEDOR_SACOLA_POSICIONADA		AND
		(LA_GERAL.di_ENV_SENS_ATU_ABERTURA_AV)			THEN
			M3_LA_ENV_Z.ABS_MOVER	:= 	LA_GERAL.coord_Z_ENVOLVEDOR_PEGA;
			passo_GIRO_SACOLA					:=	1011;
	END_IF
		
//--------------------------------------------------------------------------------------------------------------------------------------------------------------------------------
1011://se estiver rodando, libera movimento do eixo Z do Envolvedor

	IF LA_GERAL.bit_MAQUINA_RODANDO THEN
		LA_ENV.bit_EIXO_Z_ENVOLVEDOR_MOVER_ABS	:= TRUE;
		passo_GIRO_SACOLA								:= 1012;	
	END_IF
	
//--------------------------------------------------------------------------------------------------------------------------------------------------------------------------------
1012://verifica se eixo Z do Envolvedor está se movendo ou se já está posicionado

	IF	M3_LA_ENV_Z.bit_MOVE_ABS_FAZENDO OR LA_ENV.bit_EIXO_Z_ENVOLVEDOR_POSICIONADO	THEN
		LA_ENV.bit_EIXO_Z_ENVOLVEDOR_MOVER_ABS	:= FALSE;
		
		passo_GIRO_SACOLA								:= 1013;
	END_IF
	
//--------------------------------------------------------------------------------------------------------------------------------------------------------------------------------
1013://verifica se eixo Z do Envolvedor completou movimento e declara que sacola não está mais posicionada na esteira transportadora do envolvedor

	IF	M3_LA_ENV_Z.bit_MOVE_ABS_FEITO OR LA_ENV.bit_EIXO_Z_ENVOLVEDOR_POSICIONADO	THEN
	//	GVL_ENVOLVEDOR.bit_ENVOLVEDOR_SACOLA_POSICIONADA	:= FALSE;
		LA_ENV.bit_EIXO_Z_ENVOLVEDOR_MOVER_ABS		:= FALSE;
		
		passo_GIRO_SACOLA					:= 1014;
	END_IF
		
//--------------------------------------------------------------------------------------------------------------------------------------------------------------------------------
1014://se estiver rodando, aciona atuador aprox garra

	IF LA_GERAL.bit_MAQUINA_RODANDO AND LA_IHM.bit_SIMULA_GIRO THEN
		LA_ENV.bit_valv_APROX_GARRA	:=	TRUE;
		tmr_APROX_GARRA.IN					:=	TRUE;
		passo_GIRO_SACOLA					:=	1015;
	END_IF
	
//--------------------------------------------------------------------------------------------------------------------------------------------------------------------------------
1015://espera feedback do sensor de avanço do aprox garra e aciona garra dupla
	
	IF	((LA_GERAL.di_ENV_SENS_ATU_ABERTURA_RC) OR tmr_APROX_GARRA.Q) AND LA_IHM.bit_SIMULA_GIRO AND (PVAR.rec_ATUAL.int_NUM_MAX_CAMADAS_EMPILHADOR = 4) THEN
		tmr_APROX_GARRA.IN					:=	FALSE;
		tmr_GARRA_DUPLA.IN					:=	TRUE;
		passo_GIRO_SACOLA					:=	1016;
	END_IF
	
	IF	((LA_GERAL.di_ENV_SENS_ATU_ABERTURA_RC) OR tmr_APROX_GARRA.Q) AND LA_IHM.bit_SIMULA_GIRO AND (PVAR.rec_ATUAL.int_NUM_MAX_CAMADAS_EMPILHADOR = 5) THEN
		tmr_APROX_GARRA.IN					:=	FALSE;
		tmr_GARRA_DUPLA.IN					:=	TRUE;
		passo_GIRO_SACOLA					:=	1016;
	END_IF	
	
//--------------------------------------------------------------------------------------------------------------------------------------------------------------------------------
1016:	

	M3_LA_ENV_Z.ABS_MOVER.sp_POSICAO	:= 	LA_GERAL.coord_Z_ENVOLVEDOR_PEGA.sp_POSICAO + 50;
	LA_ENV.bit_EIXO_Z_ENVOLVEDOR_MOVER_ABS	:= TRUE;
	passo_GIRO_SACOLA								:= 1017;
	
//--------------------------------------------------------------------------------------------------------------------------------------------------------------------------------
1017://verifica se eixo Z do Envolvedor está se movendo ou se já está posicionado

	IF	M3_LA_ENV_Z.bit_MOVE_ABS_FAZENDO OR LA_ENV.bit_EIXO_Z_ENVOLVEDOR_POSICIONADO	THEN
		LA_ENV.bit_EIXO_Z_ENVOLVEDOR_MOVER_ABS	:= FALSE;
		LA_ENV.bit_valv_GARRA_DUPLA				:= TRUE;
		
		passo_GIRO_SACOLA								:= 1018;
	END_IF
	
//--------------------------------------------------------------------------------------------------------------------------------------------------------------------------------
1018://verifica se eixo Z do Envolvedor completou movimento e declara que sacola não está mais posicionada na esteira transportadora do envolvedor

	IF	M3_LA_ENV_Z.bit_MOVE_ABS_FEITO OR LA_ENV.bit_EIXO_Z_ENVOLVEDOR_POSICIONADO	THEN
		LA_ENV.bit_ENVOLVEDOR_SACOLA_POSICIONADA	:= FALSE;
		LA_ENV.bit_EIXO_Z_ENVOLVEDOR_MOVER_ABS		:= FALSE;
		
		passo_GIRO_SACOLA					:= 1019;
	END_IF
	
//--------------------------------------------------------------------------------------------------------------------------------------------------------------------------------
1019://espera feedback do sensor de avanço da garra dupla

	IF	(*(NOT sens_PINCA_GARRA_RC_LD AND NOT sens_PINCA_GARRA_RC_LE) OR*) tmr_GARRA_DUPLA.Q THEN
		LA_ENV.bit_valv_GARRA_DUPLA		:= TRUE;
		tmr_GARRA_DUPLA.IN						:=	FALSE;
		passo_GIRO_SACOLA						:=	1020;
	END_IF	
	
//--------------------------------------------------------------------------------------------------------------------------------------------------------------------------------
1020://	comanda posição de Saída pega do eixo Z do envolvedor e desliga vácuo filme

	IF 	LA_GERAL.bit_MAQUINA_RODANDO 				THEN
			M3_LA_ENV_Z.ABS_MOVER	:= 	LA_GERAL.coord_Z_ENVOLVEDOR_SAIDA_PEGA;
			passo_GIRO_SACOLA					:=	1021;
	END_IF
		
	
//--------------------------------------------------------------------------------------------------------------------------------------------------------------------------------
1021://se estiver rodando, libera movimento do eixo Z do Envolvedor

	IF LA_GERAL.bit_MAQUINA_RODANDO THEN
			LA_ENV.bit_EIXO_Z_ENVOLVEDOR_MOVER_ABS	:= TRUE;
			passo_GIRO_SACOLA								:= 1022;	
	END_IF
	
//--------------------------------------------------------------------------------------------------------------------------------------------------------------------------------
1022://verifica se eixo Z do Envolvedor está se movendo ou se já está posicionado

	IF	M3_LA_ENV_Z.bit_MOVE_ABS_FAZENDO OR LA_ENV.bit_EIXO_Z_ENVOLVEDOR_POSICIONADO	THEN
			LA_ENV.bit_EIXO_Z_ENVOLVEDOR_MOVER_ABS	:= FALSE;
			passo_GIRO_SACOLA								:= 1023;
	END_IF
	
//--------------------------------------------------------------------------------------------------------------------------------------------------------------------------------
1023://verifica se eixo Z do Envolvedor completou movimento

	IF	M3_LA_ENV_Z.bit_MOVE_ABS_FEITO OR LA_ENV.bit_EIXO_Z_ENVOLVEDOR_POSICIONADO	THEN
			LA_ENV.bit_EIXO_Z_ENVOLVEDOR_MOVER_ABS	:= FALSE;
			LA_ENV.bit_ENVOLVEDOR_SACOLA_POSICIONADA	:= FALSE;
			passo_GIRO_SACOLA					:= 1024;
	END_IF
	
//--------------------------------------------------------------------------------------------------------------------------------------------------------------------------------
1024://comanda eixo X do envolvedor para posição de corte de filme e eixos de giro para posição final de enrolamento de filme 
	IF LA_GERAL.bit_MAQUINA_RODANDO	THEN
			LA_ENV.bit_ENV_CORTE_FILME		:= TRUE;
			M4_LA_ENV_X.ABS_MOVER		:= LA_GERAL.coord_X_ENVOLVEDOR_CORTE;
			M5_LA_ENV_GIRO_LD.REL_MOVER	:= LA_GERAL.coord_GIRO_ENVOLVEDOR_CORTE;
			M6_LA_ENV_GIRO_LE.REL_MOVER	:= LA_GERAL.coord_GIRO_ENVOLVEDOR_CORTE;
			passo_GIRO_SACOLA 						:= 1025;
	END_IF
		
//--------------------------------------------------------------------------------------------------------------------------------------------------------------------------------
1025: //Comanda eixos X e rotativos do Envolvedor com movimentos absolutos para ponto de corte de filme. 

	LA_ENV.bit_EIXO_X_ENVOLVEDOR_MOVER_ABS				:= TRUE;
	LA_ENV.bit_EIXO_GIRO_ENVOLVEDOR_LD_MOVER_REL		:= TRUE;
	LA_ENV.bit_EIXO_GIRO_ENVOLVEDOR_LE_MOVER_REL		:= TRUE;
	passo_GIRO_SACOLA 		:= 1026;
	
//--------------------------------------------------------------------------------------------------------------------------------------------------------------------------------
1026: //Verifica se Eixo X do envolvedor está se movimentando ou se já está posicionado

	IF	M4_LA_ENV_X.bit_MOVE_ABS_FAZENDO	OR 	LA_ENV.bit_EIXO_X_ENVOLVEDOR_POSICIONADO	THEN
			LA_ENV.bit_EIXO_X_ENVOLVEDOR_MOVER_ABS	:= FALSE;
			passo_GIRO_SACOLA 								:= 1027;
	END_IF
	
//--------------------------------------------------------------------------------------------------------------------------------------------------------------------------------
1027: //Verifica se Eixo LD do envolvedor está se movimentando ou se já está posicionado

	IF	M5_LA_ENV_GIRO_LD.bit_MOVE_REL_FAZENDO	OR LA_ENV.bit_EIXO_GIRO_ENVOLVEDOR_LD_POSICIONADO	THEN
			passo_GIRO_SACOLA 				:= 1028;
	END_IF
	
//--------------------------------------------------------------------------------------------------------------------------------------------------------------------------------
1028: //Verifica se Eixo LE do envolvedor está se movimentando ou se já está posicionado

	IF	M6_LA_ENV_GIRO_LE.bit_MOVE_REL_FAZENDO		OR 	LA_ENV.bit_EIXO_GIRO_ENVOLVEDOR_LE_POSICIONADO	THEN
			passo_GIRO_SACOLA 				:= 1029;
	END_IF
	
//--------------------------------------------------------------------------------------------------------------------------------------------------------------------------------
1029: //verifica se Eixos LD, LE e X chegaram aos seus pontos

	IF	M4_LA_ENV_X.bit_MOVE_ABS_FEITO	OR 	LA_ENV.bit_EIXO_X_ENVOLVEDOR_POSICIONADO	THEN
			bit_ENTREGA_X_FEITO			:= TRUE;
	END_IF	
	
	IF	M5_LA_ENV_GIRO_LD.bit_MOVE_REL_FEITO	(*OR 	GVL_ENVOLVEDOR.bit_EIXO_GIRO_ENVOLVEDOR_LD_POSICIONADO*)	THEN
			bit_ENTREGA_GIRO_LD_FEITO	:= TRUE;
			LA_ENV.bit_EIXO_GIRO_ENVOLVEDOR_LD_MOVER_REL	:= FALSE;
	END_IF	
	
	IF	M6_LA_ENV_GIRO_LE.bit_MOVE_REL_FEITO	(*OR 	GVL_ENVOLVEDOR.bit_EIXO_GIRO_ENVOLVEDOR_LE_POSICIONADO*)	THEN
			bit_ENTREGA_GIRO_LE_FEITO	:= TRUE;
			LA_ENV.bit_EIXO_GIRO_ENVOLVEDOR_LE_MOVER_REL	:= FALSE;
	END_IF	
	
	IF	bit_ENTREGA_X_FEITO				AND
		bit_ENTREGA_GIRO_LE_FEITO		AND
		bit_ENTREGA_GIRO_LD_FEITO		THEN
			bit_ENTREGA_X_FEITO			:= FALSE;
			bit_ENTREGA_GIRO_LD_FEITO	:= FALSE;
			bit_ENTREGA_GIRO_LE_FEITO	:= FALSE;
			passo_GIRO_SACOLA 			:= 1030;
	END_IF
		
//--------------------------------------------------------------------------------------------------------------------------------------------------------------------------------
1030://	comanda posição de corte de filme do eixo Z do envolvedor

	IF 	LA_GERAL.bit_MAQUINA_RODANDO 				THEN
			LA_ENV.bit_ENV_CORTE_FILME		:= TRUE;
			M3_LA_ENV_Z.ABS_MOVER		:= LA_GERAL.coord_Z_ENVOLVEDOR_CORTE;
			M5_LA_ENV_GIRO_LD.REL_MOVER	:= LA_GERAL.coord_GIRO_ENVOLVEDOR_ENTREGA;
			M6_LA_ENV_GIRO_LE.REL_MOVER	:= LA_GERAL.coord_GIRO_ENVOLVEDOR_ENTREGA;			
			passo_GIRO_SACOLA					:=	1031;
	END_IF
		
//--------------------------------------------------------------------------------------------------------------------------------------------------------------------------------
1031://se estiver rodando, libera movimento do eixo Z do Envolvedor

	IF LA_GERAL.bit_MAQUINA_RODANDO THEN
			LA_ENV.bit_EIXO_Z_ENVOLVEDOR_MOVER_ABS			:= TRUE;
			LA_ENV.bit_EIXO_GIRO_ENVOLVEDOR_LD_MOVER_REL	:= TRUE;
			LA_ENV.bit_EIXO_GIRO_ENVOLVEDOR_LE_MOVER_REL	:= TRUE;
			passo_GIRO_SACOLA								:= 1032;	
	END_IF
	
//--------------------------------------------------------------------------------------------------------------------------------------------------------------------------------
1032://verifica se eixo Z do Envolvedor está se movendo ou se já está posicionado

	IF	M3_LA_ENV_Z.bit_MOVE_ABS_FAZENDO OR LA_ENV.bit_EIXO_Z_ENVOLVEDOR_POSICIONADO	THEN
			LA_ENV.bit_EIXO_Z_ENVOLVEDOR_MOVER_ABS		:= FALSE;
			LA_ENV.bit_EIXO_GIRO_ENVOLVEDOR_LD_MOVER_REL	:= FALSE;
			LA_ENV.bit_EIXO_GIRO_ENVOLVEDOR_LE_MOVER_REL	:= FALSE;
			passo_GIRO_SACOLA								:= 1033;
	END_IF
	
//--------------------------------------------------------------------------------------------------------------------------------------------------------------------------------
1033://verifica se eixo Z do Envolvedor completou movimento

	IF	M3_LA_ENV_Z.bit_MOVE_ABS_FEITO OR LA_ENV.bit_EIXO_Z_ENVOLVEDOR_POSICIONADO AND LA_GERAL.bit_MAQUINA_RODANDO	THEN
			LA_ENV.bit_EIXO_Z_ENVOLVEDOR_MOVER_ABS	:= FALSE;
			LA_ENV.bit_valv_VACUO_FILME	:=	TRUE;
			tmr_PASSO_1028.IN					:= TRUE;
			passo_GIRO_SACOLA					:= 1034;
	END_IF
	
	
//--------------------------------------------------------------------------------------------------------------------------------------------------------------------------------
1034://aciona valvula de corte e vácuo de filme

	IF tmr_PASSO_1028.Q	AND LA_GERAL.bit_MAQUINA_RODANDO	THEN
		tmr_PASSO_1028.IN					:= 	FALSE;
			LA_ENV.bit_valv_CORTE_FILME	:=	FALSE;
			LA_ENV.bit_ENV_CORTE_FILME	:=	FALSE;
			passo_GIRO_SACOLA					:= 	1035;
	END_IF


//--------------------------------------------------------------------------------------------------------------------------------------------------------------------------------
1035:

		M3_LA_ENV_Z.ABS_MOVER.sp_POSICAO			:=	275;
		M3_LA_ENV_Z.ABS_MOVER.sp_VELOCIDADE		:=	LA_GERAL.coord_Z_ENVOLVEDOR_ENTREGA.sp_VELOCIDADE;
		M3_LA_ENV_Z.ABS_MOVER.sp_ACELERACAO		:=	LA_GERAL.coord_Z_ENVOLVEDOR_ENTREGA.sp_ACELERACAO;
		M3_LA_ENV_Z.ABS_MOVER.sp_DESACELERACAO	:=	LA_GERAL.coord_Z_ENVOLVEDOR_ENTREGA.sp_DESACELERACAO;
		passo_GIRO_SACOLA										:=	1036;
		
//--------------------------------------------------------------------------------------------------------------------------------------------------------------------------------
1036:

	IF 	LA_GERAL.bit_MAQUINA_RODANDO	THEN
			LA_ENV.bit_EIXO_Z_ENVOLVEDOR_MOVER_ABS	:= TRUE;
			passo_GIRO_SACOLA								:= 1037;
	END_IF
	
//--------------------------------------------------------------------------------------------------------------------------------------------------------------------------------
1037://verifica se eixo Z do Envolvedor está se movendo ou se já está posicionado

	IF	M3_LA_ENV_Z.bit_MOVE_ABS_FAZENDO OR LA_ENV.bit_EIXO_Z_ENVOLVEDOR_POSICIONADO	THEN
			LA_ENV.bit_EIXO_Z_ENVOLVEDOR_MOVER_ABS	:= FALSE;
			passo_GIRO_SACOLA								:= 1038;
	END_IF
	
//--------------------------------------------------------------------------------------------------------------------------------------------------------------------------------
1038://verifica se eixo Z do Envolvedor completou movimento

	IF	M3_LA_ENV_Z.bit_MOVE_ABS_FEITO OR LA_ENV.bit_EIXO_Z_ENVOLVEDOR_POSICIONADO	THEN
			LA_ENV.bit_EIXO_Z_ENVOLVEDOR_MOVER_ABS	:= FALSE;
			passo_GIRO_SACOLA					:= 1039;
	END_IF
	
//--------------------------------------------------------------------------------------------------------------------------------------------------------------------------------
1039://espera não ter sacola depositada para comandar eixo X para Entrega
	
	IF NOT LA_ENV.bit_ENVOLVEDOR_SACOLA_DEPOSITADA	AND
		   sens_FECHA_FILME_1_RC				 			THEN
			 M4_LA_ENV_X.ABS_MOVER				:= 	LA_GERAL.coord_X_ENVOLVEDOR_ENTREGA;
			 LA_ENV.bit_ENVOLVEDOR_SACOLA_DEPOSITANDO	:=	TRUE;
			 passo_GIRO_SACOLA									:=	1040;	
	END_IF

	
//--------------------------------------------------------------------------------------------------------------------------------------------------------------------------------
1040://se estiver rodando, libera movimento do eixo X do Envolvedor

	IF LA_GERAL.bit_MAQUINA_RODANDO THEN
			LA_ENV.bit_EIXO_X_ENVOLVEDOR_MOVER_ABS	:= TRUE;
			passo_GIRO_SACOLA								:=	1041;	
	END_IF
	
//--------------------------------------------------------------------------------------------------------------------------------------------------------------------------------
1041://verifica se eixo X do Envolvedor está se movendo ou se já está posicionado

	IF	M4_LA_ENV_X.bit_MOVE_ABS_FAZENDO OR LA_ENV.bit_EIXO_X_ENVOLVEDOR_POSICIONADO	THEN
			LA_ENV.bit_EIXO_X_ENVOLVEDOR_MOVER_ABS	:= FALSE;
			passo_GIRO_SACOLA								:= 1042;
	END_IF
	
//--------------------------------------------------------------------------------------------------------------------------------------------------------------------------------
1042://verifica se eixo X do Envolvedor completou movimento

	IF	M4_LA_ENV_X.bit_MOVE_ABS_FEITO OR LA_ENV.bit_EIXO_X_ENVOLVEDOR_POSICIONADO	THEN
			LA_ENV.bit_EIXO_X_ENVOLVEDOR_MOVER_ABS	:= FALSE;
			passo_GIRO_SACOLA					:= 1043;
	END_IF
	
//--------------------------------------------------------------------------------------------------------------------------------------------------------------------------------
1043://aguarda confirmação de presença de filme para comandar eixo Z para posição de Saida Pega
	
	IF (*sens_FILME_ENVOLVEDOR AND *)LA_GERAL.bit_MAQUINA_RODANDO THEN	
			M3_LA_ENV_Z.ABS_MOVER			:=	LA_GERAL.coord_Z_ENVOLVEDOR_ENTREGA;
			passo_GIRO_SACOLA							:=	1044;
	END_IF
		
//--------------------------------------------------------------------------------------------------------------------------------------------------------------------------------
1044://se estiver rodando, libera movimento do eixo Z do Envolvedor

	IF LA_GERAL.bit_MAQUINA_RODANDO THEN
			LA_ENV.bit_EIXO_Z_ENVOLVEDOR_MOVER_ABS	:= TRUE;
			passo_GIRO_SACOLA								:= 1045;	
	END_IF
	
//--------------------------------------------------------------------------------------------------------------------------------------------------------------------------------
1045://verifica se eixo Z do Envolvedor está se movendo ou se já está posicionado

	IF	M3_LA_ENV_Z.bit_MOVE_ABS_FAZENDO OR LA_ENV.bit_EIXO_Z_ENVOLVEDOR_POSICIONADO	THEN
			LA_ENV.bit_EIXO_Z_ENVOLVEDOR_MOVER_ABS	:= FALSE;
			passo_GIRO_SACOLA								:= 1046;
	END_IF
	
//--------------------------------------------------------------------------------------------------------------------------------------------------------------------------------
1046://verifica se eixo Z do Envolvedor completou movimento

	IF	M3_LA_ENV_Z.bit_MOVE_ABS_FEITO OR LA_ENV.bit_EIXO_Z_ENVOLVEDOR_POSICIONADO	THEN
			LA_ENV.bit_EIXO_Z_ENVOLVEDOR_MOVER_ABS	:= FALSE;
			passo_GIRO_SACOLA					:= 1047;
	END_IF
	
//--------------------------------------------------------------------------------------------------------------------------------------------------------------------------------
1047://espera não ter sacola depositada para comandar eixo X para Entrega
	
	IF NOT LA_ENV.bit_ENVOLVEDOR_SACOLA_DEPOSITADA	AND
		   sens_FECHA_FILME_1_RC				 			THEN
			 M4_LA_ENV_X.ABS_MOVER				:= 	LA_GERAL.coord_X_ENVOLVEDOR_ENTREGA;
			 LA_ENV.bit_ENVOLVEDOR_SACOLA_DEPOSITANDO	:=	TRUE;
			 passo_GIRO_SACOLA									:=	1048;	
	END_IF

	
//--------------------------------------------------------------------------------------------------------------------------------------------------------------------------------
1048://se estiver rodando, libera movimento do eixo X do Envolvedor

	IF LA_GERAL.bit_MAQUINA_RODANDO THEN
			LA_ENV.bit_EIXO_X_ENVOLVEDOR_MOVER_ABS	:= TRUE;
			passo_GIRO_SACOLA								:=	1049;	
	END_IF
	
//--------------------------------------------------------------------------------------------------------------------------------------------------------------------------------
1049://verifica se eixo X do Envolvedor está se movendo ou se já está posicionado

	IF	M4_LA_ENV_X.bit_MOVE_ABS_FAZENDO OR LA_ENV.bit_EIXO_X_ENVOLVEDOR_POSICIONADO	THEN
			LA_ENV.bit_EIXO_X_ENVOLVEDOR_MOVER_ABS	:= FALSE;
			passo_GIRO_SACOLA								:= 1050;
	END_IF
	
//--------------------------------------------------------------------------------------------------------------------------------------------------------------------------------
1050://verifica se eixo X do Envolvedor completou movimento

	IF	M4_LA_ENV_X.bit_MOVE_ABS_FEITO OR LA_ENV.bit_EIXO_X_ENVOLVEDOR_POSICIONADO	THEN
			LA_ENV.bit_EIXO_X_ENVOLVEDOR_MOVER_ABS	:= FALSE;
			passo_GIRO_SACOLA					:= 1051;
	END_IF
	
	
//--------------------------------------------------------------------------------------------------------------------------------------------------------------------------------
1051://aciona fecha filme 1 e espera timer
	
	LA_ENV.bit_valv_FECHA_FILME_1	:=	TRUE;
	tmr_FECHA_FILME_1.IN					:=	TRUE;
		
	IF tmr_FECHA_FILME_1.Q	THEN
		tmr_FECHA_FILME_1.IN	:= FALSE;
		passo_GIRO_SACOLA		:= 1052;
	END_IF
	
	
//--------------------------------------------------------------------------------------------------------------------------------------------------------------------------------
1052://abre garra dupla e aciona timer
	
	LA_ENV.bit_valv_GARRA_DUPLA	:=	FALSE;
	tmr_GARRA_DUPLA2.IN					:=	TRUE;
	passo_GIRO_SACOLA					:= 1053;	
	
	
//--------------------------------------------------------------------------------------------------------------------------------------------------------------------------------
1053: //aguarda feedback dos sensores ou timer e recua atuador aprox. garra

	IF	(*(NOT sens_PINCA_GARRA_RC_LD AND NOT sens_PINCA_GARRA_RC_LE) OR*) tmr_GARRA_DUPLA2.Q THEN
			tmr_GARRA_DUPLA2.IN					:=	FALSE;
			tmr_GARRA_DUPLA3.IN					:=	TRUE;
			LA_ENV.bit_valv_APROX_GARRA	:=	FALSE;
			passo_GIRO_SACOLA					:=	1054;
	END_IF
	

//--------------------------------------------------------------------------------------------------------------------------------------------------------------------------------
1054://espera timer completar e fecha garra dupla novamente

	IF tmr_GARRA_DUPLA3.Q	THEN
			tmr_GARRA_DUPLA3.IN					:=	FALSE;
			LA_ENV.bit_valv_GARRA_DUPLA	:=	TRUE;
			passo_GIRO_SACOLA					:=	1055;
	END_IF
	
	
//--------------------------------------------------------------------------------------------------------------------------------------------------------------------------------
1055://aguarda confirmação de recuo de atuador prox. garra e confirma sacola depositada

	IF LA_GERAL.di_ENV_SENS_ATU_ABERTURA_AV THEN
			LA_ENV.bit_ENVOLVEDOR_SACOLA_DEPOSITANDO := FALSE;
			passo_GIRO_SACOLA								 :=	1056;
	END_IF
	
//--------------------------------------------------------------------------------------------------------------------------------------------------------------------------------
1056://	comanda posição de corte de filme do eixo Z do envolvedor

	IF 	LA_GERAL.bit_MAQUINA_RODANDO 				THEN
			M3_LA_ENV_Z.ABS_MOVER				 := LA_GERAL.coord_Z_ENVOLVEDOR_SAIDA_PEGA;
			passo_GIRO_SACOLA								 :=	1057;
	END_IF
		
//--------------------------------------------------------------------------------------------------------------------------------------------------------------------------------
1057://se estiver rodando, libera movimento do eixo Z do Envolvedor

	IF LA_GERAL.bit_MAQUINA_RODANDO THEN
			LA_ENV.bit_EIXO_Z_ENVOLVEDOR_MOVER_ABS	:= TRUE;
			passo_GIRO_SACOLA								:= 1058;	
	END_IF
	
//--------------------------------------------------------------------------------------------------------------------------------------------------------------------------------
1058://verifica se eixo Z do Envolvedor está se movendo ou se já está posicionado

	IF	M3_LA_ENV_Z.bit_MOVE_ABS_FAZENDO OR LA_ENV.bit_EIXO_Z_ENVOLVEDOR_POSICIONADO	THEN
			LA_ENV.bit_EIXO_Z_ENVOLVEDOR_MOVER_ABS	:= FALSE;
			passo_GIRO_SACOLA								:= 1059;
	END_IF
	
//--------------------------------------------------------------------------------------------------------------------------------------------------------------------------------
1059://verifica se eixo Z do Envolvedor completou movimento

	IF	M3_LA_ENV_Z.bit_MOVE_ABS_FEITO OR LA_ENV.bit_EIXO_Z_ENVOLVEDOR_POSICIONADO	THEN
			LA_ENV.bit_EIXO_Z_ENVOLVEDOR_MOVER_ABS	:= FALSE;
			LA_ENV.bit_ENVOLVEDOR_SACOLA_DEPOSITADA	 :=	TRUE;
			passo_GIRO_SACOLA					:= 1060;
	END_IF
	
	
//--------------------------------------------------------------------------------------------------------------------------------------------------------------------------------
1060: //reinicia ciclo comandando para posição de pega
		passo_GIRO_SACOLA				:=	999;

END_CASE


//------------//-----------LÓGICAS EXTRAS---------------//----------------------//--------------------------//


	//EIXO X ENVOLVEDOR JÁ ESTÁ NA POSIÇÃO
	IF	LA_ENV.info_MOTOR_X_ENVOLVEDOR_POS_ATUAL	>= M4_LA_ENV_X.ABS_MOVER.sp_POSICAO - 1	AND
		LA_ENV.info_MOTOR_X_ENVOLVEDOR_POS_ATUAL	<= M4_LA_ENV_X.ABS_MOVER.sp_POSICAO + 1	THEN
			LA_ENV.bit_EIXO_X_ENVOLVEDOR_POSICIONADO	:= TRUE;
	ELSE
			LA_ENV.bit_EIXO_X_ENVOLVEDOR_POSICIONADO	:= FALSE;
	END_IF
	
	//EIXO Z ENVOLVEDOR JÁ ESTÁ NA POSIÇÃO
	IF	LA_ENV.info_MOTOR_Z_ENVOLVEDOR_POS_ATUAL	>= M3_LA_ENV_Z.ABS_MOVER.sp_POSICAO - 1	AND
		LA_ENV.info_MOTOR_Z_ENVOLVEDOR_POS_ATUAL	<= M3_LA_ENV_Z.ABS_MOVER.sp_POSICAO + 1	THEN
			LA_ENV.bit_EIXO_Z_ENVOLVEDOR_POSICIONADO	:= TRUE;
	ELSE
			LA_ENV.bit_EIXO_Z_ENVOLVEDOR_POSICIONADO	:= FALSE;
	END_IF
	
	//EIXO GIRO LD ENVOLVEDOR JÁ ESTÁ NA POSIÇÃO
	IF	LA_ENV.info_MOTOR_GIRO_ENVOLVIMENTO_LD_POS_ATUAL	>= M5_LA_ENV_GIRO_LD.ABS_MOVER.sp_POSICAO - 1	AND
		LA_ENV.info_MOTOR_GIRO_ENVOLVIMENTO_LD_POS_ATUAL	<= M5_LA_ENV_GIRO_LD.ABS_MOVER.sp_POSICAO + 1	THEN
			LA_ENV.bit_EIXO_GIRO_ENVOLVEDOR_LD_POSICIONADO	:= TRUE;
	ELSE
			LA_ENV.bit_EIXO_GIRO_ENVOLVEDOR_LD_POSICIONADO	:= FALSE;
	END_IF
	
	
	//EIXO GIRO LE ENVOLVEDOR JÁ ESTÁ NA POSIÇÃO
	IF	LA_ENV.info_MOTOR_GIRO_ENVOLVIMENTO_LE_POS_ATUAL	>= M6_LA_ENV_GIRO_LE.ABS_MOVER.sp_POSICAO - 1	AND
		LA_ENV.info_MOTOR_GIRO_ENVOLVIMENTO_LE_POS_ATUAL	<= M6_LA_ENV_GIRO_LE.ABS_MOVER.sp_POSICAO + 1	THEN
			LA_ENV.bit_EIXO_GIRO_ENVOLVEDOR_LE_POSICIONADO	:= TRUE;
	ELSE
			LA_ENV.bit_EIXO_GIRO_ENVOLVEDOR_LE_POSICIONADO	:= FALSE;
	END_IF



//-----------ATUADORES-------------//--------------------//---------------------//

LA_GERAL.do_ENV_ATU_GARRAS		:=	NOT LA_ENV.bit_valv_GARRA_DUPLA;
LA_GERAL.do_ENV_ATU_ABERTURA	:=	 NOT LA_ENV.bit_valv_APROX_GARRA;

valv_CORTE_FILME				:=	LA_ENV.bit_valv_CORTE_FILME;
valv_VACUO_FILME				:=	LA_ENV.bit_valv_VACUO_FILME;
LA_GERAL.do_ENV_CORTE_FILME		:=	(LA_ENV.bit_ENV_CORTE_FILME AND LA_GERAL.bit_SAFETY_ATIVO) OR LA_IHM.bit_ENV_CORTE_FILME;
	
	
tmr_GARRA_DUPLA(PT:= T#500MS);
tmr_GARRA_DUPLA2(PT:= T#100MS);
tmr_GARRA_DUPLA3(PT:= T#50MS);
tmr_APROX_GARRA(PT:= T#1800MS);
tmr_FECHA_FILME_1(PT:= T#1800MS);

tmr_PASSO_1028(PT:= T#1000MS);
tmr_PASSO_1029(PT:= T#1500MS);

END_PROGRAM

// LADO_A/03 - LA_ENVOLVEDOR/C02_MANUAL
PROGRAM C02_MANUAL
VAR
	rtrig_EIXO_Z_ENVOLVEDOR_RESET_STOP			: R_TRIG;
	rtrig_EIXO_x_ENVOLVEDOR_RESET_STOP			: R_TRIG;
	rtrig_EIXO_GIRO_ENVOLVEDOR_LD_RESET_STOP	: R_TRIG;
	rtrig_EIXO_GIRO_ENVOLVEDOR_LE_RESET_STOP	: R_TRIG;
	
	bit_EIXO_Z_ENVOLVEDOR_RTRIG					: BOOL;
	bit_EIXO_X_ENVOLVEDOR_RTRIG					: BOOL;
	bit_EIXO_GIRO_ENVOLVEDOR_LD_RTRIG			: BOOL;
	bit_EIXO_GIRO_ENVOLVEDOR_LE_RTRIG			: BOOL;
END_VAR

//MODO MANUAL EIXOS


	//EIXO Z ENVOLVEDOR
	IF		LA_IHM.bit_MANUAL_HABILITAR_EIXOS							AND
		NOT	LA_ENV.bit_MOTOR_Z_ENVOLVEDOR_JOG_FORWARD			AND	
		NOT	LA_ENV.bit_MOTOR_Z_ENVOLVEDOR_JOG_REVERSE			THEN
				bit_EIXO_Z_ENVOLVEDOR_RTRIG	:= TRUE;
	ELSE
				bit_EIXO_Z_ENVOLVEDOR_RTRIG	:= FALSE;
	END_IF
	
	rtrig_EIXO_Z_ENVOLVEDOR_RESET_STOP(CLK := bit_EIXO_Z_ENVOLVEDOR_RTRIG);
	LA_ENV.bit_MOTOR_Z_ENVOLVEDOR_JOG_STOP	:= rtrig_EIXO_Z_ENVOLVEDOR_RESET_STOP.Q;


	//EIXO X ENVOLVEDOR
	IF		LA_IHM.bit_MANUAL_HABILITAR_EIXOS							AND
		NOT	LA_ENV.bit_MOTOR_X_ENVOLVEDOR_JOG_FORWARD			AND	
		NOT	LA_ENV.bit_MOTOR_X_ENVOLVEDOR_JOG_REVERSE			THEN
				bit_EIXO_X_ENVOLVEDOR_RTRIG	:= TRUE;
	ELSE
				bit_EIXO_X_ENVOLVEDOR_RTRIG	:= FALSE;
	END_IF
	
	rtrig_EIXO_x_ENVOLVEDOR_RESET_STOP(CLK := bit_EIXO_X_ENVOLVEDOR_RTRIG);
	LA_ENV.bit_MOTOR_X_ENVOLVEDOR_JOG_STOP	:= rtrig_EIXO_x_ENVOLVEDOR_RESET_STOP.Q;
	
	

	//EIXO LD 
	IF		LA_IHM.bit_MANUAL_HABILITAR_EIXOS							AND
		NOT	LA_ENV.bit_MOTOR_GIRO_ENVOLVEDOR_LD_JOG_FORWARD		AND	
		NOT	LA_ENV.bit_MOTOR_GIRO_ENVOLVEDOR_LD_JOG_REVERSE		THEN
				bit_EIXO_GIRO_ENVOLVEDOR_LD_RTRIG	:= TRUE;
	ELSE
				bit_EIXO_GIRO_ENVOLVEDOR_LD_RTRIG	:= FALSE;
	END_IF
	
	rtrig_EIXO_GIRO_ENVOLVEDOR_LD_RESET_STOP(CLK := bit_EIXO_GIRO_ENVOLVEDOR_LD_RTRIG);
	LA_ENV.bit_MOTOR_GIRO_ENVOLVEDOR_LD_JOG_STOP	:= rtrig_EIXO_GIRO_ENVOLVEDOR_LD_RESET_STOP.Q;
	
	
	//EIXO LE
	IF		LA_IHM.bit_MANUAL_HABILITAR_EIXOS							AND
		NOT	LA_ENV.bit_MOTOR_GIRO_ENVOLVEDOR_LE_JOG_FORWARD		AND	
		NOT	LA_ENV.bit_MOTOR_GIRO_ENVOLVEDOR_LE_JOG_REVERSE		THEN
				bit_EIXO_GIRO_ENVOLVEDOR_LE_RTRIG	:= TRUE;
	ELSE
				bit_EIXO_GIRO_ENVOLVEDOR_LE_RTRIG	:= FALSE;
	END_IF
	
	rtrig_EIXO_GIRO_ENVOLVEDOR_LE_RESET_STOP(CLK := bit_EIXO_GIRO_ENVOLVEDOR_LE_RTRIG);
	LA_ENV.bit_MOTOR_GIRO_ENVOLVEDOR_LE_JOG_STOP	:= rtrig_EIXO_GIRO_ENVOLVEDOR_LE_RESET_STOP.Q;
	
//--------------------------//-----------------------------------//---------------------------//--------------------------------//	
	
//HOME DOS EIXOS

	//HOME EIXO Z ENVOLVEDOR
	IF	(LA_ENV.bit_EIXO_Z_ENVOLVEDOR_FAZER_HOME OR LA_IHM.bit_EIXO_Z_ENVOLVEDOR_FAZER_HOME)	THEN
			M3_LA_ENV_Z.bit_FAZER_HOME	:= TRUE;
	END_IF
	
	IF	M3_LA_ENV_Z.bit_HOME_FEITO		THEN
			M3_LA_ENV_Z.bit_FAZER_HOME	:= FALSE;
	END_IF
	
	//HOME EIXO X ENVOLVEDOR
	IF	(LA_ENV.bit_EIXO_X_ENVOLVEDOR_FAZER_HOME OR LA_IHM.bit_EIXO_X_ENVOLVEDOR_FAZER_HOME)	THEN
			M4_LA_ENV_X.bit_FAZER_HOME	:= TRUE;
	END_IF
	
	IF	M3_LA_ENV_Z.bit_HOME_FEITO		THEN
			M4_LA_ENV_X.bit_FAZER_HOME	:= FALSE;
	END_IF


	//HOME EIXO LD ENVOLVEDOR
	IF	(LA_ENV.bit_EIXO_GIRO_ENVOLVEDOR_LD_FAZER_HOME OR LA_IHM.bit_EIXO_GIRO_ENVOLVEDOR_LD_FAZER_HOME)	THEN
			M5_LA_ENV_GIRO_LD.bit_FAZER_HOME	:= TRUE;
	END_IF
	
	IF	M5_LA_ENV_GIRO_LD.bit_HOME_FEITO		THEN
			M5_LA_ENV_GIRO_LD.bit_FAZER_HOME	:= FALSE;
	END_IF
	
	
	
	//HOME EIXO LE ENVOLVEDOR
	IF	(LA_ENV.bit_EIXO_GIRO_ENVOLVEDOR_LE_FAZER_HOME OR LA_IHM.bit_EIXO_GIRO_ENVOLVEDOR_LE_FAZER_HOME)	THEN
			M6_LA_ENV_GIRO_LE.bit_FAZER_HOME	:= TRUE;
	END_IF
	
	IF	M1_LA_EMP_GARRA.bit_HOME_FEITO		THEN
			M6_LA_ENV_GIRO_LE.bit_FAZER_HOME	:= FALSE;
	END_IF

END_PROGRAM

// LADO_A/03 - LA_ENVOLVEDOR/C03_EST_ENTRADA
PROGRAM C03_EST_ENTRADA
VAR
	passo_EST_ENTRADA	: INT := 9;
	RESET_ROTINA		: BOOL;
	
	f_trig_SENS_ENTRADA : F_TRIG;
	tmr_PARAR_ESTEIRA	: TON;
END_VAR

IF LA_IHM.bit_bt_RESET_EST_ENTRADA	THEN
	 passo_EST_ENTRADA := 9;
END_IF



CASE passo_EST_ENTRADA OF
	
//--------------------------------------------------------------------------------------------------------------------------------------------------------------------------------
09: //RESET VARIAVEIS

	//caso não há presença de sacola no sensor, declara que a esteira está cheia
	IF sens_EST_TRANS_PRESENCA THEN
		LA_ENV.bit_EST_ENTRADA_CHEIA	:= TRUE;
		passo_EST_ENTRADA 						:= 999;
	ELSE
		LA_ENV.bit_EST_ENTRADA_CHEIA	:=	FALSE;
		passo_EST_ENTRADA := 998;
	END_IF
	
	
//--------------------------------------------------------------------------------------------------------------------------------------------------------------------------------
998://Prepara para iniciar ciclo e liga esteira

	LA_ENV.est_ENTRADA_ENVOLVEDOR	:=	true;
	passo_EST_ENTRADA 						:= 	999;
	
	
//--------------------------------------------------------------------------------------------------------------------------------------------------------------------------------
999://se houver pilha de sacola no final da esteira, declara que está com esteira de entrada do envolvedor cheia para impedir que mesa de giro libere roletes
	//se não houver pilha de sacola na esteira transportadora, deixa esteira ligada

	
	IF NOT 	LA_ENV.bit_ENVOLVEDOR_SACOLA_POSICIONADA AND 
			LA_GERAL.bit_MAQUINA_RODANDO 					 AND 
			LA_EMP.bit_ENTREGANDO_PILHA_COMPLETA   THEN
				LA_ENV.est_ENTRADA_ENVOLVEDOR	:=	TRUE;
				passo_EST_ENTRADA 						:= 	1000;
	END_IF
	
	
	
//--------------------------------------------------------------------------------------------------------------------------------------------------------------------------------
1000:

	IF LA_ENV.bit_ENVOLVEDOR_SACOLA_POSICIONADA AND sens_EST_TRANS_PRESENCA THEN
		LA_ENV.est_ENTRADA_ENVOLVEDOR	:=	FALSE;
	ELSE
		LA_ENV.est_ENTRADA_ENVOLVEDOR	:=	TRUE;
	END_IF
	
	
	IF f_trig_SENS_ENTRADA.Q THEN
		tmr_PARAR_ESTEIRA.IN					:=	TRUE;
		passo_EST_ENTRADA 						:= 	1001;
	END_IF
	
	
	
//--------------------------------------------------------------------------------------------------------------------------------------------------------------------------------
1001:

	IF tmr_PARAR_ESTEIRA.Q	AND LA_GERAL.bit_MAQUINA_RODANDO	THEN
		tmr_PARAR_ESTEIRA.IN					:=	FALSE;
		LA_ENV.est_ENTRADA_ENVOLVEDOR	:=	FALSE;	
		passo_EST_ENTRADA 						:= 	999;
	END_IF



END_CASE


	IF sens_EST_TRANS_PRESENCA THEN
		LA_ENV.bit_EST_ENTRADA_CHEIA	:=	TRUE;
	ELSE
		LA_ENV.bit_EST_ENTRADA_CHEIA	:=	FALSE;
	END_IF
	
	tmr_PARAR_ESTEIRA(PT:= T#500MS);
	f_trig_SENS_ENTRADA(CLK:= sens_EST_TRANS_PRESENCA);

END_PROGRAM

// LADO_A/03 - LA_ENVOLVEDOR/C04_EST_TRANSPORTADOR
PROGRAM C04_EST_TRANSPORTADOR
VAR
	passo_EST_TRANSPORTADOR	:	INT	:=	9;
	tmr_PILHA_POSICIONADA	: 	TON;
	RESET_ROTINA			: 	BOOL;
END_VAR

IF LA_IHM.bit_bt_RESET_EST_TR	THEN
	 passo_EST_TRANSPORTADOR := 9;
END_IF



CASE passo_EST_TRANSPORTADOR OF

//--------------------------------------------------------------------------------------------------------------------------------------------------------------------------------
09: //RESET VARIAVEIS

	//caso não há presença de sacola no sensor, declara que a pilha de sacolas está posicionada
	IF sens_POS_1_ENVOLVEDOR AND sens_POS_2_ENVOLVEDOR AND LA_GERAL.bit_SAFETY_ATIVO THEN
		LA_ENV.bit_ENVOLVEDOR_SACOLA_POSICIONADA	:= TRUE;
	ELSE
		LA_ENV.bit_ENVOLVEDOR_SACOLA_POSICIONADA	:= FALSE;
	END_IF
	
	passo_EST_TRANSPORTADOR 							:= 999;
	
	
//--------------------------------------------------------------------------------------------------------------------------------------------------------------------------------
999://se pilha de sacola estiver posicionada, declara que está posicionada para garra pegar e desliga esteira. Se não, mantém ela ligada

	(*IF sens_POS_2_ENVOLVEDOR (*AND sens_POS_2_ENVOLVEDOR sens_FILME_ENVOLVEDOR*) THEN
		//GVL_ENVOLVEDOR.est_TRANSPORTADOR_ENVOLVEDOR			:=	FALSE;
		tmr_PILHA_POSICIONADA.IN							:= 	TRUE;
	ELSE
		GVL_ENVOLVEDOR.est_TRANSPORTADOR_ENVOLVEDOR			:=	TRUE;
	END_IF
	
	IF tmr_PILHA_POSICIONADA.Q	THEN
		GVL_ENVOLVEDOR.bit_ENVOLVEDOR_SACOLA_POSICIONADA	:=	TRUE;
		GVL_ENVOLVEDOR.est_TRANSPORTADOR_ENVOLVEDOR			:=	FALSE;
		passo_EST_TRANSPORTADOR								:= 	1000;
	END_IF*)
	
	IF sens_POS_1_ENVOLVEDOR AND LA_GERAL.bit_MAQUINA_RODANDO THEN	
		tmr_PILHA_POSICIONADA.IN							:= 	TRUE;
	ELSE
		LA_ENV.est_TRANSPORTADOR_ENVOLVEDOR			:=	TRUE;
	END_IF
	
	IF tmr_PILHA_POSICIONADA.Q	THEN
		LA_ENV.bit_ENVOLVEDOR_SACOLA_POSICIONADA	:=	TRUE;
		LA_ENV.est_TRANSPORTADOR_ENVOLVEDOR			:=	FALSE;
		LA_ENV.est_TRANSPORTADOR_ENVOLVEDOR			:=	FALSE;
		passo_EST_TRANSPORTADOR								:= 	1000;
	END_IF
	
	
//--------------------------------------------------------------------------------------------------------------------------------------------------------------------------------
1000://após confirmação de que a sacola não está mais posicionada, liga esteira e reinicia ciclo

	tmr_PILHA_POSICIONADA.IN	:=	FALSE;

	IF NOT LA_ENV.bit_ENVOLVEDOR_SACOLA_POSICIONADA THEN
		LA_ENV.est_TRANSPORTADOR_ENVOLVEDOR			:=	TRUE;
		passo_EST_TRANSPORTADOR								:= 	999;
	END_IF



END_CASE



//tmr_PILHA_POSICIONADA(PT:= T#1355MS);//pilha 40x50
//tmr_PILHA_POSICIONADA(PT:= T#1325MS);//pilha 36x48
tmr_PILHA_POSICIONADA(PT:= T#18MS);//pilha 50x60

END_PROGRAM

// LADO_A/03 - LA_ENVOLVEDOR/C05_EST_SAIDA
PROGRAM C05_EST_SAIDA
VAR
	reset_rotina	:	BOOL;
	tmr_PASSO_1001	:	TON;
	tmr_PASSO_1003	:	TON;
	tmr_PASSO_1007	:	TON;
	tmr_PASSO_1010	:	TON;
	passo_EST_SAIDA	:	INT := 9;
END_VAR

IF LA_IHM.bit_bt_RESET_EST_SAIDA THEN
	passo_EST_SAIDA	:=	9;	
END_IF


CASE passo_EST_SAIDA OF
	
//--------------------------------------------------------------------------------------------------------------------------------------------------------------------------------
09: //HOME: Reseta variáveis e recua atuadores
	
	LA_ENV.bit_valv_FECHA_FILME_1	:=	FALSE;
	LA_ENV.bit_valv_FECHA_FILME_2	:=	FALSE;
	LA_ENV.bit_valv_FECHA_FILME_3	:=	FALSE;
	LA_ENV.est_SAIDA_ENVOLVEDOR		:=	FALSE;
	
	LA_ENV.bit_ENVOLVEDOR_SACOLA_DEPOSITADA	:=	FALSE;
	LA_ENV.bit_ENVOLVEDOR_ENVIANDO_PILHA	:=	FALSE;
	
	tmr_PASSO_1001.IN						:=	FALSE;
	tmr_PASSO_1003.IN						:= FALSE;
	tmr_PASSO_1007.IN						:=	FALSE;
	tmr_PASSO_1010.IN						:= FALSE;
	passo_EST_SAIDA	:=	10;
	
//--------------------------------------------------------------------------------------------------------------------------------------------------------------------------------
10:	//aguarda feedback dos sensores de recuo dos atuadores

	IF 	sens_FECHA_FILME_1_RC	AND
		sens_FECHA_FILME_2_RC	AND
		sens_FECHA_FILME_3_RC	THEN
			passo_EST_SAIDA	:=	999;
	END_IF	
	
	
//--------------------------------------------------------------------------------------------------------------------------------------------------------------------------------
999: //inicio de ciclo com máquina rodando

	IF LA_GERAL.bit_MAQUINA_RODANDO	THEN
		passo_EST_SAIDA	:=	1000;
	END_IF
	
	
//--------------------------------------------------------------------------------------------------------------------------------------------------------------------------------
1000: //aguarda confirmação de pilha de sacola depositada na esteira de saida e recua fecha filme 1

	IF 	LA_ENV.bit_ENVOLVEDOR_SACOLA_DEPOSITADA 	(*OR 
   (NOT GVL_ENVOLVEDOR.bit_ENVOLVEDOR_SACOLA_DEPOSITANDO	AND
		sens_SAIDA_ENVOLVEDOR_1) 	*)						THEN
			LA_ENV.bit_valv_FECHA_FILME_1	:=	FALSE;
			passo_EST_SAIDA	:=	1001;
	END_IF
	
	
//--------------------------------------------------------------------------------------------------------------------------------------------------------------------------------
1001://espera feedback do sensor de recuo do fecha filme 1, e liga esteira

	IF sens_FECHA_FILME_1_RC AND LA_GERAL.bit_MAQUINA_RODANDO THEN
		tmr_PASSO_1001.IN	:=	TRUE;
	END_IF
	
	IF tmr_PASSO_1001.Q	THEN
		LA_ENV.est_SAIDA_ENVOLVEDOR	:=	TRUE;
		passo_EST_SAIDA						:=	1002;
		tmr_PASSO_1001.IN					:=	FALSE;
	END_IF
	
	
//--------------------------------------------------------------------------------------------------------------------------------------------------------------------------------
1002://assim que chegar no sensor de saida do envolvedor 2, desliga esteira

	IF sens_SAIDA_ENVOLVEDOR_2 THEN
		LA_ENV.est_SAIDA_ENVOLVEDOR	:=	FALSE;
		passo_EST_SAIDA	:=	1003;
	END_IF
	
//--------------------------------------------------------------------------------------------------------------------------------------------------------------------------------
1003://aciona atuador fecha filme 2

	IF LA_GERAL.bit_MAQUINA_RODANDO THEN
		LA_ENV.bit_valv_FECHA_FILME_2	:=	TRUE;
		tmr_PASSO_1003.IN := TRUE;
		passo_EST_SAIDA	:=	1004;
	END_IF
	
	
//--------------------------------------------------------------------------------------------------------------------------------------------------------------------------------
1004://espera confirmaçao de avanço e recua atuador fecha filme 2

	IF tmr_PASSO_1003.Q AND LA_GERAL.bit_MAQUINA_RODANDO THEN
		tmr_PASSO_1003.IN := FALSE;
		LA_ENV.bit_valv_FECHA_FILME_2	:=	FALSE;
		passo_EST_SAIDA	:=	1005;
	END_IF
	
//--------------------------------------------------------------------------------------------------------------------------------------------------------------------------------
1005://espera confirmação de recuo e liga esteira
	
	IF sens_FECHA_FILME_2_RC AND LA_GERAL.bit_MAQUINA_RODANDO THEN
		LA_ENV.est_SAIDA_ENVOLVEDOR	:=	TRUE;
		passo_EST_SAIDA	:=	1006;
	END_IF
	
	
//--------------------------------------------------------------------------------------------------------------------------------------------------------------------------------
1006://assim que chegar no sensor de saida do envolvedor 3, desliga esteira

	IF sens_SAIDA_ENVOLVEDOR_3 THEN
		LA_ENV.est_SAIDA_ENVOLVEDOR	:=	FALSE;
		passo_EST_SAIDA	:=	1007;
	END_IF
	
	
//--------------------------------------------------------------------------------------------------------------------------------------------------------------------------------
1007://aciona atuador fecha filme 3

	IF LA_GERAL.bit_MAQUINA_RODANDO	THEN
		LA_ENV.bit_valv_FECHA_FILME_3	:=	TRUE;
		tmr_PASSO_1007.IN						:= TRUE;
		passo_EST_SAIDA	:=	1008;
	END_IF
	
	
//--------------------------------------------------------------------------------------------------------------------------------------------------------------------------------
1008://aguarda confirmação de avanço de atuador fecha filme 3

	IF (*sens_FECHA_FILME_3_AV AND*) tmr_PASSO_1007.Q	THEN
		tmr_PASSO_1007.IN						:=	FALSE;
		LA_ENV.bit_valv_FECHA_FILME_3	:=	FALSE;
		passo_EST_SAIDA	:=	1009;
	END_IF
	
	
//--------------------------------------------------------------------------------------------------------------------------------------------------------------------------------
1009://aguarda confirmação de recuo de atuador fecha filme 3 e liga esteira

	IF sens_FECHA_FILME_3_RC	THEN
		//GVL_ENVOLVEDOR.est_SAIDA_ENVOLVEDOR	:=	TRUE;
		passo_EST_SAIDA	:=	1011;
	END_IF
	
//--------------------------------------------------------------------------------------------------------------------------------------------------------------------------------
1010://Caso atinja o sensor de saida da esteira do envolvedor 4, e não esteja no processo de pesar sacola e o atuador de transferencia esteja avançado, pula para próximo passo. Se não, desliga esteira
	
	
	IF 	sens_SAIDA_ENVOLVEDOR_4 AND (NOT GVL_PESAGEM.bit_PESANDO_PILHA_SACOLA OR NOT sens_TRANSFERENCIA_AV)	THEN
			LA_ENV.est_SAIDA_ENVOLVEDOR	:=	FALSE;
			tmr_PASSO_1010.IN					:=	TRUE;
			passo_EST_SAIDA						:=	1011;
	END_IF
	
	
//--------------------------------------------------------------------------------------------------------------------------------------------------------------------------------
1011:

	IF 	NOT GVL_PESAGEM.bit_PESANDO_PILHA_SACOLA AND sens_TRANSFERENCIA_AV (*AND tmr_PASSO_1010.Q*)	THEN
			LA_ENV.est_SAIDA_ENVOLVEDOR			 :=	TRUE;
			LA_ENV.bit_ENVOLVEDOR_ENVIANDO_PILHA :=	TRUE;
			tmr_PASSO_1010.IN							 := false;
			passo_EST_SAIDA								 :=	1012;
	END_IF
	
	
//--------------------------------------------------------------------------------------------------------------------------------------------------------------------------------
1012://aguarda pilha de sacola sair da esteira para desligar esteira

	IF sens_MESA_TRANSFER_1 OR sens_MESA_TRANSFER_2	THEN
		LA_ENV.est_SAIDA_ENVOLVEDOR				:=	FALSE;
		LA_ENV.bit_ENVOLVEDOR_SACOLA_DEPOSITADA	:=	FALSE;
		LA_ENV.bit_ENVOLVEDOR_ENVIANDO_PILHA 	:=	FALSE;
		passo_EST_SAIDA	:=	999;
	END_IF
	
	







END_CASE




//------------//-----------LÓGICAS EXTRAS---------------//----------------------//--------------------------//

//-----------ATUADORES-------------//--------------------//---------------------//

valv_FECHA_FILME_1		:=	LA_ENV.bit_valv_FECHA_FILME_1;
valv_FECHA_FILME_2		:=	LA_ENV.bit_valv_FECHA_FILME_2;
valv_FECHA_FILME_3		:=	LA_ENV.bit_valv_FECHA_FILME_3;



//-----------RETOMADA--------------//------------------//---------------------//

(*IF GVL_ENVOLVEDOR.bit_ENVOLVEDOR_SACOLA_DEPOSITADA AND reset_rotina THEN
	IF 	passo_EST_SAIDA >= 999 	AND
			passo_EST_SAIDA <= 1001	THEN
			
			passo_EST_SAIDA := 999;
		END_IF
	
		IF 	passo_EST_SAIDA >= 1002 AND
			passo_EST_SAIDA <= 1005	THEN
			
			passo_EST_SAIDA := 1002;
		END_IF	
	
		IF 	passo_EST_SAIDA >= 1006 AND
			passo_EST_SAIDA <= 1009	THEN
			
			passo_EST_SAIDA := 1006;
	END_IF
ELSIF NOT GVL_ENVOLVEDOR.bit_ENVOLVEDOR_SACOLA_DEPOSITADA AND reset_rotina	THEN
			passo_EST_SAIDA := 9;
END_IF
	
*)

tmr_PASSO_1001(PT:= T#300MS);
tmr_PASSO_1003(PT:= T#2500MS);
tmr_PASSO_1007(PT:= T#3000MS);
tmr_PASSO_1010(PT:= T#10000MS);

END_PROGRAM

// LADO_A/03 - LA_ENVOLVEDOR/C06_ENTRADAS_REMOTAS
PROGRAM C06_ENTRADAS_REMOTAS
VAR
END_VAR

END_PROGRAM

// LADO_A/03 - LA_ENVOLVEDOR/C07_SAIDAS_REMOTAS
PROGRAM C07_SAIDAS_REMOTAS
VAR
END_VAR

END_PROGRAM

// LADO_A/05 - LA_IHM/E00_TELA_RECEITAS
PROGRAM E00_TELA_RECEITAS
VAR
	tmr_STATUS_RECEITA			: TON;
END_VAR


//BOTÃO CARREGAR: Move a receita selecionada da lista de receitas para ser mostrada na tela
	IF	LA_IHM.bt_CARREGAR_RECEITA	THEN
			LA_GERAL.rec_IHM	:= PVAR.RECEITAS[LA_IHM.int_RECEITA_ATUAL];
			LA_IHM.int_STATUS_RECEITA	:= 1;
	END_IF
	
//BOTÃO SALVAR: Move a receita que está sendo mostrada na tela para a receita selecionada da lista de receitas
	IF	LA_IHM.bt_SALVAR_RECEITA	THEN
			PVAR.RECEITAS[LA_IHM.int_RECEITA_ATUAL] := LA_GERAL.rec_IHM;
			LA_IHM.int_STATUS_RECEITA	:= 2;
	END_IF
	
//BOTÃO UPLOAD: Move a receita que está atualmente sendo executada para ser mostrada na tela
	IF	LA_IHM.bt_UPLOAD_RECEITA	THEN
			LA_GERAL.rec_IHM	:= PVAR.rec_ATUAL;
			LA_IHM.int_STATUS_RECEITA	:= 3;
	END_IF
	
//BOTÃO DOWNLOAD: Move a receita que está sendo mostrada na tela para a que será executada
	IF	LA_IHM.bt_DOWNLOAD_RECEITA	THEN
			PVAR.rec_ATUAL	:= LA_GERAL.rec_IHM;
			LA_IHM.int_STATUS_RECEITA	:= 4;
	END_IF
	
//STATUS RECEITA
	IF tmr_STATUS_RECEITA.Q		THEN
			LA_IHM.int_STATUS_RECEITA	:= 0;
	END_IF
		
//RECEITA SELECIONADA
	LA_GERAL.rec_SELECIONADA	:= PVAR.RECEITAS[LA_IHM.int_RECEITA_ATUAL];
	
//SELECAO DO MODO DE OPERAÇÃO
		
(*	IF GVL_IHM.bit_SELEC_MODO_2	THEN
			GVL_IHM.int_RECEITA_QNTD_CORES := 2;
	END_IF
	
	IF GVL_IHM.bit_SELEC_MODO_3	THEN
			GVL_IHM.int_RECEITA_QNTD_CORES := 3;
	END_IF
	
	IF GVL_IHM.bit_SELEC_MODO_4	THEN
			GVL_IHM.int_RECEITA_QNTD_CORES := 4;
	END_IF*)
		
//SELECAO DE RECEITA PARA DUAS CORES
		IF	LA_IHM.bit_SELEC_RECEITA_1	THEN	
				LA_IHM.int_RECEITA_ATUAL	:= 1;
		END_IF
		
		IF	LA_IHM.bit_SELEC_RECEITA_2	THEN	
				LA_IHM.int_RECEITA_ATUAL	:= 2;
		END_IF
		
		IF	LA_IHM.bit_SELEC_RECEITA_3	THEN	
				LA_IHM.int_RECEITA_ATUAL	:= 3;
		END_IF
		
		IF	LA_IHM.bit_SELEC_RECEITA_4	THEN	
				LA_IHM.int_RECEITA_ATUAL	:= 4;
		END_IF
		
		IF	LA_IHM.bit_SELEC_RECEITA_5	THEN	
				LA_IHM.int_RECEITA_ATUAL	:= 5;
		END_IF
		
		IF	LA_IHM.bit_SELEC_RECEITA_6	THEN	
				LA_IHM.int_RECEITA_ATUAL	:= 6;
		END_IF
		
		IF	LA_IHM.bit_SELEC_RECEITA_7	THEN	
				LA_IHM.int_RECEITA_ATUAL	:= 7;
		END_IF
		
		IF	LA_IHM.bit_SELEC_RECEITA_8	THEN	
				LA_IHM.int_RECEITA_ATUAL	:= 8;
		END_IF
		
		IF	LA_IHM.bit_SELEC_RECEITA_9	THEN	
				LA_IHM.int_RECEITA_ATUAL	:= 9;
		END_IF
		
		IF	LA_IHM.bit_SELEC_RECEITA_10	THEN	
				LA_IHM.int_RECEITA_ATUAL	:= 10;
		END_IF
	
	
//NOMES DAS RECEITAS
				LA_IHM.nome_RECEITA_1	:= PVAR.RECEITAS[1].NOME;
				LA_IHM.nome_RECEITA_2	:= PVAR.RECEITAS[2].NOME;
				LA_IHM.nome_RECEITA_3	:= PVAR.RECEITAS[3].NOME;
				LA_IHM.nome_RECEITA_4	:= PVAR.RECEITAS[4].NOME;
				LA_IHM.nome_RECEITA_5	:= PVAR.RECEITAS[5].NOME;
				LA_IHM.nome_RECEITA_6	:= PVAR.RECEITAS[6].NOME;
				LA_IHM.nome_RECEITA_7	:= PVAR.RECEITAS[7].NOME;
				LA_IHM.nome_RECEITA_8	:= PVAR.RECEITAS[8].NOME;
				LA_IHM.nome_RECEITA_9	:= PVAR.RECEITAS[9].NOME;
				LA_IHM.nome_RECEITA_10	:= PVAR.RECEITAS[10].NOME;
		
	
//================================================================================================================================================================================
//TIMERS
tmr_STATUS_RECEITA (IN:= (NOT LA_IHM.bt_CARREGAR_RECEITA AND NOT LA_IHM.bt_SALVAR_RECEITA AND NOT LA_IHM.bt_UPLOAD_RECEITA AND NOT LA_IHM.bt_DOWNLOAD_RECEITA), PT:= T#5S);

END_PROGRAM

// LADO_A/05 - LA_IHM/E01_TELA_ATUADORES_EMPILHADOR
PROGRAM E01_TELA_ATUADORES_EMPILHADOR
VAR
END_VAR

//SE A MÁQUINA ESTIVER EM MODO MANUAL E NÃO ESTIVER RODANDO, HABILITA SELEÇÃO MANUAL DE ATUADORES
	IF	LA_GERAL.bit_MAQUINA_MANUAL	AND
	NOT	LA_GERAL.bit_MAQUINA_RODANDO	THEN
			
			IF LA_IHM.bit_SELEC_EMPILHADOR_BANDEJA			THEN
					LA_IHM.int_EMPILHADOR_ATUADOR_SELECIONADO	:= 1;
			END_IF
			
			
			IF LA_IHM.bit_SELEC_EMPILHADOR_DESCE_MESA_GIRO		THEN
					LA_IHM.int_EMPILHADOR_ATUADOR_SELECIONADO	:= 2;
			END_IF
			
			IF LA_IHM.bit_SELEC_EMPILHADOR_GARRA_SACOLA		THEN
					LA_IHM.int_EMPILHADOR_ATUADOR_SELECIONADO	:= 3;
			END_IF
			
			IF LA_IHM.bit_SELEC_EMPILHADOR_POSICIONA_SACOLA		THEN
					LA_IHM.int_EMPILHADOR_ATUADOR_SELECIONADO	:= 4;
			END_IF

		
			
			CASE	LA_IHM.int_EMPILHADOR_ATUADOR_SELECIONADO	OF
					
					0: //SEM ATUADOR SELECIONADO
						LA_IHM.bit_ATU_EMPILHADOR_AVANCADO	:= FALSE;
						LA_IHM.bit_ATU_EMPILHADOR_RECUADO	:= FALSE;			
			
					1://ATUADOR EMPILHADOR BANDEJA
						IF LA_IHM.bit_ATU_EMPILHADOR_AVANCAR	THEN
								LA_EMP.bit_valv_BANDEJA	:= TRUE;
						END_IF
						
						IF LA_IHM.bit_ATU_EMPILHADOR_RECUAR	THEN
								LA_EMP.bit_valv_BANDEJA	:= FALSE;
						END_IF
						
						LA_IHM.bit_ATU_EMPILHADOR_AVANCADO	:= LA_EMP.di_SENS_APOIO_BANDEJA_AV;
						LA_IHM.bit_ATU_EMPILHADOR_RECUADO	:= LA_EMP.di_SENS_APOIO_BANDEJA_RC;
						
					2://ATUADOR DESCE GIRO MESA
						IF LA_IHM.bit_ATU_EMPILHADOR_AVANCAR	THEN
								LA_EMP.bit_valv_DESCE_MESA_GIRO	:= TRUE;
						END_IF
						
						IF LA_IHM.bit_ATU_EMPILHADOR_RECUAR	THEN
								LA_EMP.bit_valv_DESCE_MESA_GIRO	:= FALSE;
						END_IF
						
						LA_IHM.bit_ATU_EMPILHADOR_AVANCADO	:= LA_EMP.di_SENS_MESA_GIRO_AV;
						LA_IHM.bit_ATU_EMPILHADOR_RECUADO	:= LA_EMP.di_SENS_MESA_GIRO_RC;
						
					3://ATUADOR GARRA SACOLA
						IF LA_IHM.bit_ATU_EMPILHADOR_AVANCAR	THEN
								LA_EMP.bit_valv_GARRA_SACOLA	:= TRUE;
						END_IF
						
						IF LA_IHM.bit_ATU_EMPILHADOR_RECUAR	THEN
								LA_EMP.bit_valv_GARRA_SACOLA	:= FALSE;
						END_IF
						
						LA_IHM.bit_ATU_EMPILHADOR_AVANCADO	:= LA_EMP.di_SENS_PINCA_GARRA_EMPILHADOR_AV;
						LA_IHM.bit_ATU_EMPILHADOR_RECUADO	:= LA_EMP.di_SENS_PINCA_GARRA_EMPILHADOR_RC;
						
					4://ATUADOR POSICIONA SACOLA
						IF LA_IHM.bit_ATU_EMPILHADOR_AVANCAR	THEN
								LA_EMP.bit_valv_POSICIONA_SACOLA	:= TRUE;
						END_IF
						
						IF LA_IHM.bit_ATU_EMPILHADOR_RECUAR	THEN
								LA_EMP.bit_valv_POSICIONA_SACOLA	:= FALSE;
						END_IF
						
						LA_IHM.bit_ATU_EMPILHADOR_AVANCADO	:= sens_POSICIONADOR_EMPILHADOR_AV;
						LA_IHM.bit_ATU_EMPILHADOR_RECUADO	:= sens_POSICIONADOR_EMPILHADOR_RC;					
		
			END_CASE	
	
	ELSE
		
		LA_IHM.int_EMPILHADOR_ATUADOR_SELECIONADO	:= 0;
		
		LA_IHM.bit_ATU_EMPILHADOR_AVANCADO				:= FALSE;
		LA_IHM.bit_ATU_EMPILHADOR_RECUADO				:= FALSE;	
			
		LA_IHM.bit_SELEC_EMPILHADOR_BANDEJA			:= FALSE;
		LA_IHM.bit_SELEC_EMPILHADOR_DESCE_MESA_GIRO 	:= FALSE;
		LA_IHM.bit_SELEC_EMPILHADOR_GARRA_SACOLA	 	:= FALSE;
		LA_IHM.bit_SELEC_EMPILHADOR_POSICIONA_SACOLA	:= FALSE;

	
	END_IF

END_PROGRAM

// LADO_A/05 - LA_IHM/E02_TELA_ATUADORES_ENVOLVEDOR
PROGRAM E02_TELA_ATUADORES_ENVOLVEDOR
VAR
END_VAR

//SE A MÁQUINA ESTIVER EM MODO MANUAL E NÃO ESTIVER RODANDO, HABILITA SELEÇÃO MANUAL DE ATUADORES
	IF	LA_GERAL.bit_MAQUINA_MANUAL	AND
	NOT	LA_GERAL.bit_MAQUINA_RODANDO	THEN
			
			IF LA_IHM.bit_SELEC_ENVOLVEDOR_APROX_GARRA		THEN
					LA_IHM.int_ENVOLVEDOR_ATUADOR_SELECIONADO	:= 1;
			END_IF
			
			
			IF LA_IHM.bit_SELEC_ENVOLVEDOR_GARRA_DUPLA		THEN
					LA_IHM.int_ENVOLVEDOR_ATUADOR_SELECIONADO	:= 2;
			END_IF
			
			IF LA_IHM.bit_SELEC_ENVOLVEDOR_CORTE_FILME		THEN
					LA_IHM.int_ENVOLVEDOR_ATUADOR_SELECIONADO	:= 3;
			END_IF
			
			IF LA_IHM.bit_SELEC_ENVOLVEDOR_VACUO_FILME		THEN
					LA_IHM.int_ENVOLVEDOR_ATUADOR_SELECIONADO	:= 4;
			END_IF
			
			IF LA_IHM.bit_SELEC_ENVOLVEDOR_FECHA_FILME_1		THEN
					LA_IHM.int_ENVOLVEDOR_ATUADOR_SELECIONADO	:= 5;
			END_IF
			
			IF LA_IHM.bit_SELEC_ENVOLVEDOR_FECHA_FILME_2		THEN
					LA_IHM.int_ENVOLVEDOR_ATUADOR_SELECIONADO	:= 6;
			END_IF
			
			IF LA_IHM.bit_SELEC_ENVOLVEDOR_FECHA_FILME_3		THEN
					LA_IHM.int_ENVOLVEDOR_ATUADOR_SELECIONADO	:= 7;
			END_IF

		
			
			CASE	LA_IHM.int_ENVOLVEDOR_ATUADOR_SELECIONADO	OF
					
					0: //SEM ATUADOR SELECIONADO
						LA_IHM.bit_ATU_ENVOLVEDOR_AVANCADO	:= FALSE;
						LA_IHM.bit_ATU_ENVOLVEDOR_RECUADO	:= FALSE;			
			
					1://ATUADOR ENVOLVEDOR APROX GARRA
						IF LA_IHM.bit_ATU_ENVOLVEDOR_AVANCAR	THEN
								LA_ENV.bit_valv_APROX_GARRA	:= FALSE;
						END_IF
						
						IF LA_IHM.bit_ATU_ENVOLVEDOR_RECUAR	THEN
								LA_ENV.bit_valv_APROX_GARRA	:= TRUE;
						END_IF
						
						LA_IHM.bit_ATU_ENVOLVEDOR_AVANCADO	:= (LA_GERAL.di_ENV_SENS_ATU_ABERTURA_AV);
						LA_IHM.bit_ATU_ENVOLVEDOR_RECUADO	:= (LA_GERAL.di_ENV_SENS_ATU_ABERTURA_RC);
						
					2://ATUADOR ENVOLVEDOR GARRA DUPLA
						IF LA_IHM.bit_ATU_ENVOLVEDOR_AVANCAR	THEN
								LA_ENV.bit_valv_GARRA_DUPLA	:= FALSE;
						END_IF
						
						IF LA_IHM.bit_ATU_ENVOLVEDOR_RECUAR	THEN
								LA_ENV.bit_valv_GARRA_DUPLA	:= TRUE;
						END_IF
						
						//GVL_IHM.bit_ATU_ENVOLVEDOR_AVANCADO	:= sens_MESA_GIRO_AV;
						LA_IHM.bit_ATU_ENVOLVEDOR_RECUADO	:= LA_GERAL.di_ENV_SENS_ATU_GARRA_LD_RC AND LA_GERAL.di_ENV_SENS_ATU_GARRA_LE_RC;
						
					3://ATUADOR CORTE FILME
						IF LA_IHM.bit_ATU_ENVOLVEDOR_AVANCAR	THEN
								LA_ENV.bit_valv_CORTE_FILME	:= TRUE;
						END_IF
						
						IF LA_IHM.bit_ATU_ENVOLVEDOR_RECUAR	THEN
								LA_ENV.bit_valv_CORTE_FILME	:= FALSE;
						END_IF
						
						LA_IHM.bit_ATU_ENVOLVEDOR_AVANCADO	:= sens_CORTE_FILME_AV;
						LA_IHM.bit_ATU_ENVOLVEDOR_RECUADO	:= sens_CORTE_FILME_RC;
						
					4://ATUADOR VACUO FILME
						IF LA_IHM.bit_ATU_ENVOLVEDOR_AVANCAR	THEN
								LA_ENV.bit_valv_VACUO_FILME	:= TRUE;
						END_IF
						
						IF LA_IHM.bit_ATU_ENVOLVEDOR_RECUAR	THEN
								LA_ENV.bit_valv_VACUO_FILME	:= FALSE;
						END_IF
						
						//GVL_IHM.bit_ATU_ENVOLVEDOR_AVANCADO	:= sens_PINCA_GARRA_EMPILHADOR_AV;
						//GVL_IHM.bit_ATU_ENVOLVEDOR_RECUADO	:= sens_PINCA_GARRA_EMPILHADOR_RC;	

					5://ATUADOR FECHA FILME 1
						IF LA_IHM.bit_ATU_ENVOLVEDOR_AVANCAR	THEN
								LA_ENV.bit_valv_FECHA_FILME_1	:= TRUE;
						END_IF
						
						IF LA_IHM.bit_ATU_ENVOLVEDOR_RECUAR	THEN
								LA_ENV.bit_valv_FECHA_FILME_1	:= FALSE;
						END_IF
						
					//	GVL_IHM.bit_ATU_ENVOLVEDOR_AVANCADO	:= NOT sens_FECHA_FILME_1_RC;
						LA_IHM.bit_ATU_ENVOLVEDOR_RECUADO	:= sens_FECHA_FILME_1_RC;	

					 6://ATUADOR FECHA FILME 2
						IF LA_IHM.bit_ATU_ENVOLVEDOR_AVANCAR	THEN
								LA_ENV.bit_valv_FECHA_FILME_2	:= TRUE;
						END_IF
						
						IF LA_IHM.bit_ATU_ENVOLVEDOR_RECUAR	THEN
								LA_ENV.bit_valv_FECHA_FILME_2	:= FALSE;
						END_IF
						
						LA_IHM.bit_ATU_ENVOLVEDOR_AVANCADO	:= sens_FECHA_FILME_2_AV;
						LA_IHM.bit_ATU_ENVOLVEDOR_RECUADO	:= sens_FECHA_FILME_2_RC;	

					7://ATUADOR FECHA FILME 3
						IF LA_IHM.bit_ATU_ENVOLVEDOR_AVANCAR	THEN
								LA_ENV.bit_valv_FECHA_FILME_3	:= TRUE;
						END_IF
						
						IF LA_IHM.bit_ATU_ENVOLVEDOR_RECUAR	THEN
								LA_ENV.bit_valv_FECHA_FILME_3	:= FALSE;
						END_IF
						
						LA_IHM.bit_ATU_ENVOLVEDOR_AVANCADO	:= sens_FECHA_FILME_3_AV;
						LA_IHM.bit_ATU_ENVOLVEDOR_RECUADO	:= sens_FECHA_FILME_3_RC;				
		
			END_CASE	
	
	ELSE
		
		LA_IHM.int_ENVOLVEDOR_ATUADOR_SELECIONADO	:= 0;
		
		LA_IHM.bit_ATU_ENVOLVEDOR_AVANCADO			:= FALSE;
		LA_IHM.bit_ATU_ENVOLVEDOR_RECUADO			:= FALSE;	
			
		LA_IHM.bit_SELEC_ENVOLVEDOR_APROX_GARRA	:= FALSE;
		LA_IHM.bit_SELEC_ENVOLVEDOR_GARRA_DUPLA 	:= FALSE;
		LA_IHM.bit_SELEC_ENVOLVEDOR_CORTE_FILME	:= FALSE;
		LA_IHM.bit_SELEC_ENVOLVEDOR_VACUO_FILME	:= FALSE;
		LA_IHM.bit_SELEC_ENVOLVEDOR_FECHA_FILME_1	:= FALSE;
		LA_IHM.bit_SELEC_ENVOLVEDOR_FECHA_FILME_2	:= FALSE;
		LA_IHM.bit_SELEC_ENVOLVEDOR_FECHA_FILME_3	:= FALSE;

	
	END_IF

END_PROGRAM

// LADO_A/05 - LA_IHM/E03_TELA_ATUADORES_PESAGEM
PROGRAM E03_TELA_ATUADORES_PESAGEM
VAR
END_VAR

//SE A MÁQUINA ESTIVER EM MODO MANUAL E NÃO ESTIVER RODANDO, HABILITA SELEÇÃO MANUAL DE ATUADORES
	IF	LA_GERAL.bit_MAQUINA_MANUAL	AND
	NOT	LA_GERAL.bit_MAQUINA_RODANDO	THEN
			
			IF LA_IHM.bit_SELEC_PESAGEM_ACIONAMENTO_TRANSFERENCIA		THEN
					LA_IHM.int_PESAGEM_ATUADOR_SELECIONADO	:= 1;
			END_IF

		
			
			CASE	LA_IHM.int_PESAGEM_ATUADOR_SELECIONADO	OF
					
					0: //SEM ATUADOR SELECIONADO
						LA_IHM.bit_ATU_PESAGEM_AVANCADO	:= FALSE;
						LA_IHM.bit_ATU_PESAGEM_RECUADO		:= FALSE;			
			
					1://ATUADOR ENVOLVEDOR APROX GARRA
						IF LA_IHM.bit_ATU_PESAGEM_AVANCAR	THEN
								GVL_PESAGEM.bit_valv_ACIONAMENTO_TRANSFERENCIA	:= TRUE;
						END_IF
						
						IF LA_IHM.bit_ATU_PESAGEM_RECUAR	THEN
								GVL_PESAGEM.bit_valv_ACIONAMENTO_TRANSFERENCIA	:= FALSE;
						END_IF
						
						LA_IHM.bit_ATU_PESAGEM_AVANCADO	:= sens_TRANSFERENCIA_AV;
						LA_IHM.bit_ATU_PESAGEM_RECUADO		:= sens_TRANSFERENCIA_RC;
							
		
			END_CASE	
	
	ELSE
		
		LA_IHM.int_PESAGEM_ATUADOR_SELECIONADO				:= 0;
		
		LA_IHM.bit_ATU_PESAGEM_AVANCADO					:= FALSE;
		LA_IHM.bit_ATU_PESAGEM_RECUADO						:= FALSE;	
			
		LA_IHM.bit_SELEC_PESAGEM_ACIONAMENTO_TRANSFERENCIA	:= FALSE;
	
	END_IF

END_PROGRAM

// LADO_A/05 - LA_IHM/E04_TELA_OPERACAO
PROGRAM E04_TELA_OPERACAO
VAR
	teste	:	REAL;
END_VAR

//Espelhamento de Variaveis
	
	LA_GERAL.bit_MAQUINA_MANUAL		:= LA_IHM.bit_MAQUINA_MANUAL;
	
	LA_IHM.array_HIST_ERRO_PESAGEM_1	:=	GVL_PESAGEM.array_HIST_PESO.0;
	LA_IHM.array_HIST_ERRO_PESAGEM_2	:=	GVL_PESAGEM.array_HIST_PESO.1;
	LA_IHM.array_HIST_ERRO_PESAGEM_3	:=	GVL_PESAGEM.array_HIST_PESO.2;
	LA_IHM.array_HIST_ERRO_PESAGEM_4	:=	GVL_PESAGEM.array_HIST_PESO.3;
	LA_IHM.array_HIST_ERRO_PESAGEM_5	:=	GVL_PESAGEM.array_HIST_PESO.4;
	LA_IHM.array_HIST_ERRO_PESAGEM_6	:=	GVL_PESAGEM.array_HIST_PESO.5;
	LA_IHM.array_HIST_ERRO_PESAGEM_7	:=	GVL_PESAGEM.array_HIST_PESO.6;



	//MOTOR EIXO X EMPILHAMENTO
	IF	M0_LA_EMP_X.bit_POWER_ERRO		OR
		M0_LA_EMP_X.bit_HOME_ERRO			OR
		M0_LA_EMP_X.bit_MOVE_ABS_ERRO		OR
		M0_LA_EMP_X.bit_MOVE_REL_ERRO		OR
		EIXO_X_EMPILHADOR.bError						THEN
			LA_IHM.bit_EIXO_X_EMPILHADOR_ALARME_ATIVO	:= TRUE;
	ELSE
			LA_IHM.bit_EIXO_X_EMPILHADOR_ALARME_ATIVO	:= FALSE;	
	END_IF


	//MOTOR PEGA SACOLA
	IF	M1_LA_EMP_GARRA.bit_POWER_ERRO			OR
		M1_LA_EMP_GARRA.bit_HOME_ERRO			OR
		M1_LA_EMP_GARRA.bit_MOVE_ABS_ERRO		OR
		M1_LA_EMP_GARRA.bit_MOVE_REL_ERRO		OR
		EIXO_GARRA_EMPILHADOR.bError					THEN
			LA_IHM.bit_EIXO_GARRA_EMPILHADOR_ALARME_ATIVO	:= TRUE;
	ELSE
			LA_IHM.bit_EIXO_GARRA_EMPILHADOR_ALARME_ATIVO	:= FALSE;	
	END_IF
	
	
	//MOTOR MESA GIRO
	IF	M2_LA_EMP_GIRO.bit_POWER_ERRO			OR
		M2_LA_EMP_GIRO.bit_HOME_ERRO				OR
		M2_LA_EMP_GIRO.bit_MOVE_ABS_ERRO			OR
		M2_LA_EMP_GIRO.bit_MOVE_REL_ERRO			OR
		EIXO_GIRO_MESA.bError					THEN
			LA_IHM.bit_EIXO_GIRO_MESA_ALARME_ATIVO	:= TRUE;
	ELSE
			LA_IHM.bit_EIXO_GIRO_MESA_ALARME_ATIVO	:= FALSE;	
	END_IF
	
	
	//MOTOR EIXO Z ENVOLVEDOR
	IF	M3_LA_ENV_Z.bit_POWER_ERRO			OR
		M3_LA_ENV_Z.bit_HOME_ERRO				OR
		M3_LA_ENV_Z.bit_MOVE_ABS_ERRO			OR
		M3_LA_ENV_Z.bit_MOVE_REL_ERRO			OR
		EIXO_Z_ENVOLVEDOR.bError							THEN
			LA_IHM.bit_EIXO_Z_ENVOLVEDOR_ALARME_ATIVO	:= TRUE;
	ELSE
			LA_IHM.bit_EIXO_Z_ENVOLVEDOR_ALARME_ATIVO	:= FALSE;	
	END_IF
	
	
	//MOTOR EIXO X ENVOLVEDOR
	IF	M4_LA_ENV_X.bit_POWER_ERRO			OR
		M4_LA_ENV_X.bit_HOME_ERRO				OR
		M4_LA_ENV_X.bit_MOVE_ABS_ERRO			OR
		M4_LA_ENV_X.bit_MOVE_REL_ERRO			OR
		EIXO_X_ENVOLVEDOR.bError							THEN
			LA_IHM.bit_EIXO_X_ENVOLVEDOR_ALARME_ATIVO	:= TRUE;
	ELSE
			LA_IHM.bit_EIXO_X_ENVOLVEDOR_ALARME_ATIVO	:= FALSE;	
	END_IF
	
	
		//MOTOR GIRO ENVOLVEDOR LD
	IF	M5_LA_ENV_GIRO_LD.bit_POWER_ERRO			OR
		M5_LA_ENV_GIRO_LD.bit_HOME_ERRO			OR
		M5_LA_ENV_GIRO_LD.bit_MOVE_ABS_ERRO		OR
		M5_LA_ENV_GIRO_LD.bit_MOVE_REL_ERRO		OR
		EIXO_GIRO_ENVOLVEDOR_LD.bError								THEN
			LA_IHM.bit_EIXO_GIRO_ENVOLVEDOR_LD_ALARME_ATIVO	:= TRUE;
	ELSE
			LA_IHM.bit_EIXO_GIRO_ENVOLVEDOR_LD_ALARME_ATIVO	:= FALSE;	
	END_IF
	
		//MOTOR GIRO ENVOLVEDOR LE
	IF	M6_LA_ENV_GIRO_LE.bit_POWER_ERRO			OR
		M6_LA_ENV_GIRO_LE.bit_HOME_ERRO			OR
		M6_LA_ENV_GIRO_LE.bit_MOVE_ABS_ERRO		OR
		M6_LA_ENV_GIRO_LE.bit_MOVE_REL_ERRO		OR
		EIXO_GIRO_ENVOLVEDOR_LE.bError								THEN
			LA_IHM.bit_EIXO_GIRO_ENVOLVEDOR_LE_ALARME_ATIVO	:= TRUE;
	ELSE
			LA_IHM.bit_EIXO_GIRO_ENVOLVEDOR_LE_ALARME_ATIVO	:= FALSE;	
	END_IF
	
	
//HABILITADO
	LA_IHM.bit_EIXO_X_EMPILHADOR_HABILITADO			:= EIXO_X_EMPILHADOR.bDriveStartRealState;
	LA_IHM.bit_EIXO_GARRA_EMPILHADOR_HABILITADO		:= EIXO_GARRA_EMPILHADOR.bDriveStartRealState;
	LA_IHM.bit_EIXO_GIRO_MESA_HABILITADO				:= EIXO_GIRO_MESA.bDriveStartRealState;
	LA_IHM.bit_EIXO_Z_ENVOLVEDOR_HABILITADO			:= EIXO_Z_ENVOLVEDOR.bDriveStartRealState;
	LA_IHM.bit_EIXO_X_ENVOLVEDOR_HABILITADO			:= EIXO_X_ENVOLVEDOR.bDriveStartRealState;
	LA_IHM.bit_EIXO_GIRO_ENVOLVEDOR_LD_HABILITADO		:= EIXO_GIRO_ENVOLVEDOR_LD.bDriveStartRealState;
	LA_IHM.bit_EIXO_GIRO_ENVOLVEDOR_LE_HABILITADO		:= EIXO_GIRO_ENVOLVEDOR_LD.bDriveStartRealState;
	
//FAZENDO HOME
	LA_IHM.bit_EIXO_X_EMPILHADOR_FAZENDO_HOME			:= M0_LA_EMP_X.bit_HOME_FAZENDO;
	LA_IHM.bit_EIXO_GARRA_EMPILHADOR_FAZENDO_HOME		:= M1_LA_EMP_GARRA.bit_HOME_FAZENDO;
	LA_IHM.bit_EIXO_GIRO_MESA_FAZENDO_HOME				:= M2_LA_EMP_GIRO.bit_HOME_FAZENDO;
	LA_IHM.bit_EIXO_Z_ENVOLVEDOR_FAZENDO_HOME			:= M3_LA_ENV_Z.bit_HOME_FAZENDO;
	LA_IHM.bit_EIXO_X_ENVOLVEDOR_FAZENDO_HOME			:= M4_LA_ENV_X.bit_HOME_FAZENDO;
	LA_IHM.bit_EIXO_GIRO_ENVOLVEDOR_LD_FAZENDO_HOME	:= M5_LA_ENV_GIRO_LD.bit_HOME_FAZENDO;
	LA_IHM.bit_EIXO_GIRO_ENVOLVEDOR_LE_FAZENDO_HOME	:= M6_LA_ENV_GIRO_LE.bit_HOME_FAZENDO;
	
//POSIÇÃO ATUAL IHM
	LA_IHM.info_MANI_POS_ATUAL_X_EMPILHADOR		:=	LA_EMP.info_MOTOR_EIXO_X_EMPILHADOR_POS_ATUAL;
	LA_IHM.info_MANI_POS_ATUAL_GARRA_EMPILHADOR	:=	LA_EMP.info_MOTOR_GARRA_EMPILHADOR_POS_ATUAL;
	LA_IHM.info_MANI_POS_ATUAL_GIRO_MESA			:=	LA_EMP.info_MOTOR_GIRO_MESA_POS_ATUAL;
	LA_IHM.info_MANI_POS_ATUAL_Z_ENVOLVEDOR		:=	LA_ENV.info_MOTOR_Z_ENVOLVEDOR_POS_ATUAL;
	LA_IHM.info_MANI_POS_ATUAL_X_ENVOLVEDOR		:=	LA_ENV.info_MOTOR_X_ENVOLVEDOR_POS_ATUAL; 
	LA_IHM.info_POS_ATUAL_GIRO_EMPILHADOR_LD		:=	LA_ENV.info_MOTOR_GIRO_ENVOLVIMENTO_LD_POS_ATUAL;
	LA_IHM.info_POS_ATUAL_GIRO_EMPILHADOR_LE		:=	LA_ENV.info_MOTOR_GIRO_ENVOLVIMENTO_LE_POS_ATUAL;
	
//ALARMES ESTEIRAS
	LA_IHM.bit_feedback_ERRO_MESA_GIRO				:=	LA_EMP.di_feedback_ERRO_MESA_GIRO;
	LA_IHM.bit_feedback_ERRO_EST_INSPECAO			:=	LA_EMP.di_feedback_ERRO_EST_INSPECAO;
	LA_IHM.bit_feedback_ERRO_ENTRADA_ENVOLVEDOR	:=	feedback_ERRO_ENTRADA_ENVOLVEDOR;
	LA_IHM.bit_feedback_ERRO_TRANSP_SAIDA_1		:=	feedback_ERRO_TRANSP_SAIDA_1;
	LA_IHM.bit_feedback_ERRO_MESA_TRANSFER			:=	feedback_ERRO_MESA_TRANSFER;
	LA_IHM.bit_feedback_ERRO_REJEITO_PRODUTO		:=	feedback_ERRO_REJEITO_PRODUTO;
	LA_IHM.bit_feedback_ERRO_ESTAGIO_1				:=	feedback_ERRO_ESTAGIO_1;
	LA_IHM.bit_feedback_ERRO_MERGER_1				:=	feedback_ERRO_MERGER_1;
	
	
	
	//MÁQUINA MANUAL
IF LA_GERAL.bit_MAQUINA_MANUAL AND NOT LA_GERAL.bit_MAQUINA_PRONTA THEN

	//COMANDO DE JOG MANUAIS DOS EIXOS	
		LA_EMP.bit_EIXO_X_EMPILHADOR_JOG_FORWARD 	:=	LA_IHM.bit_EIXO_X_EMPILHADOR_JOG_POSITIVO;
		LA_EMP.bit_EIXO_X_EMPILHADOR_JOG_REVERSE 	:=	LA_IHM.bit_EIXO_X_EMPILHADOR_JOG_NEGATIVO;	
	
		LA_EMP.bit_GARRA_EMPILHADOR_JOG_FORWARD 	:=	LA_IHM.bit_EIXO_GARRA_EMPILHADOR_JOG_POSITIVO;
		LA_EMP.bit_GARRA_EMPILHADOR_JOG_REVERSE 	:=	LA_IHM.bit_EIXO_GARRA_EMPILHADOR_JOG_NEGATIVO;
		
		LA_EMP.bit_GIRO_MESA_JOG_FORWARD 			:=	LA_IHM.bit_EIXO_GIRO_MESA_JOG_POSITIVO;
		LA_EMP.bit_GIRO_MESA_JOG_REVERSE 			:=	LA_IHM.bit_EIXO_GIRO_MESA_JOG_NEGATIVO;
		
		LA_ENV.bit_MOTOR_Z_ENVOLVEDOR_JOG_FORWARD 	:=	LA_IHM.bit_EIXO_Z_ENVOLVEDOR_JOG_POSITIVO;
		LA_ENV.bit_MOTOR_Z_ENVOLVEDOR_JOG_REVERSE 	:=	LA_IHM.bit_EIXO_Z_ENVOLVEDOR_JOG_NEGATIVO;
		
		LA_ENV.bit_MOTOR_X_ENVOLVEDOR_JOG_FORWARD 	:=	LA_IHM.bit_EIXO_X_ENVOLVEDOR_JOG_POSITIVO;
		LA_ENV.bit_MOTOR_X_ENVOLVEDOR_JOG_REVERSE 	:=	LA_IHM.bit_EIXO_X_ENVOLVEDOR_JOG_NEGATIVO;
		
		LA_ENV.bit_MOTOR_GIRO_ENVOLVEDOR_LD_JOG_FORWARD 	:=	LA_IHM.bit_EIXO_GIRO_ENVOLVEDOR_LD_JOG_POSITIVO;
		LA_ENV.bit_MOTOR_GIRO_ENVOLVEDOR_LD_JOG_REVERSE 	:=	LA_IHM.bit_EIXO_GIRO_ENVOLVEDOR_LD_JOG_NEGATIVO;
		
		LA_ENV.bit_MOTOR_GIRO_ENVOLVEDOR_LE_JOG_FORWARD 	:=	LA_IHM.bit_EIXO_GIRO_ENVOLVEDOR_LE_JOG_POSITIVO;
		LA_ENV.bit_MOTOR_GIRO_ENVOLVEDOR_LE_JOG_REVERSE 	:=	LA_IHM.bit_EIXO_GIRO_ENVOLVEDOR_LE_JOG_NEGATIVO;
		
		
END_IF

END_PROGRAM

// LADO_A/05 - LA_IHM/E05_CONTADORES
PROGRAM E05_CONTADORES
VAR
	tmr_MINUTOS		: TON;
	tmr_TURNO_TROCADO : TON;
	LIM_HORA_TURNO1				: LIMITALARM;
	LIM_HORA_TURNO2				: LIMITALARM;
	LIM_HORA_TURNO3				: LIMITALARM;
	
	teste_dia					: BOOL;
	teste_reset_turno			: BOOL;
	teste_reset_cont_turnoa		: BOOL;
	
	tmr_TEMPO_RODANDO_T1		: DINT;
	tmr_TEMPO_TOTAL_T1			: LREAL;
	tmr_TEMPO_RODANDO_T2		: DINT;
	tmr_TEMPO_TOTAL_T2			: LREAL;
	tmr_TEMPO_RODANDO_T3		: DINT;
	tmr_TEMPO_TOTAL_T3			: LREAL;
	
	teste: BOOL;
END_VAR

	//CALCULOS
	//	GVL_IHM.num_CAIXAS_MEDIA		:= (GVL_MOVE.num_CAIXAS_MINUTO_MEDIA);
	//	GVL_IHM.num_CAIXAS_TOTAL		:= (GVL_MOVE.num_CAIXAS_MINUTO_TOTAL);		
	//	GVL_IHM.num_PALLETS_TOTAL		:= (GVL_MOVE.num_GERAL_PALLETS_TOTAL);

		
tmr_MINUTOS							(PT := T#60S);

LEITURA_DATA_PLC();

//================================================================================================================================================================================
//================================================================================================================================================================================
//DEFINIÇÃO DE TURNO

	//TURNO A
	IF LIM_HORA_TURNO1.IL THEN
		LA_IHM.turno_A	:=	TRUE;
		LA_IHM.turno_B	:=	FALSE;
		LA_IHM.turno_C	:=	FALSE;
	ELSE
		LA_IHM.turno_A	:=	FALSE;
	END_IF
	
	//TURNO B
	IF LIM_HORA_TURNO2.IL THEN
		LA_IHM.turno_A	:=	FALSE;
		LA_IHM.turno_B	:=	TRUE;
		LA_IHM.turno_C	:=	FALSE;
	ELSE
		LA_IHM.turno_B	:=	FALSE;
	END_IF
	
	//TURNO C
	IF NOT (LIM_HORA_TURNO3.O AND LIM_HORA_TURNO3.U) THEN
		LA_IHM.turno_A	:=	FALSE;
		LA_IHM.turno_B	:=	FALSE;
		LA_IHM.turno_C	:=	TRUE;
	ELSE
		LA_IHM.turno_C	:=	FALSE;
	END_IF
	
	//RESET TURNOS
	IF 	(LA_IHM.HORARIO_ATUAL_SEGUNDO = 57 	AND
 		LA_IHM.HORARIO_ATUAL_MINUTO = 59 		AND
		LA_IHM.HORARIO_ATUAL_HORA = 5)			OR
		teste_reset_turno			 			THEN
			LA_IHM.turno_A	:=	FALSE;
			LA_IHM.turno_B	:=	FALSE;
			LA_IHM.turno_C	:=	FALSE;
	END_IF
	


//================================================================================================================================================================================
//================================================================================================================================================================================
//CONTAGEM DO TEMPO

	//MINUTO COMPLETO
	IF LA_IHM.HORARIO_ATUAL_SEGUNDO = 59 THEN
		LA_IHM.bit_HORARIO_MINUTO_COMPLETO	:=	TRUE;
	ELSE
		LA_IHM.bit_HORARIO_MINUTO_COMPLETO	:=	FALSE;
	END_IF
	
